KUKA KRL program: MyProgram_088().src

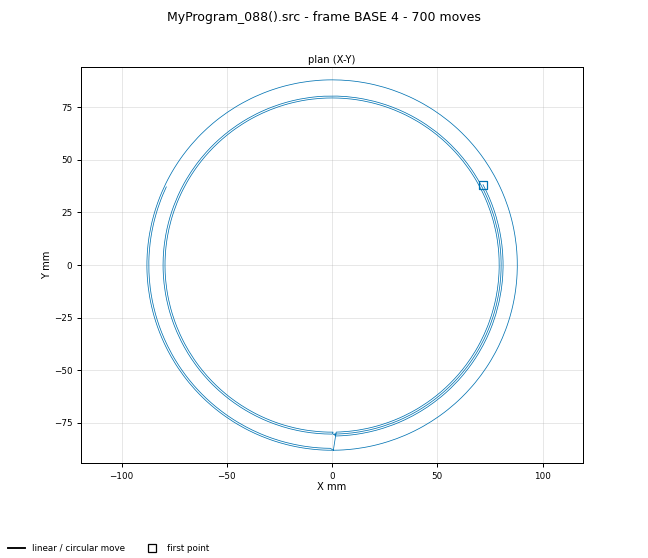
[picture p0: tool path of MyProgram_088().src in frame BASE 4, 700 of 700 moves have a stored position in this frame; points joined in program order, loops and branches not executed]
&ACCESS RVP
&REL 1
&PARAM TEMPLATE = C:\KRC\Roboter\Template\vorgabe
&PARAM EDITMASK = *
DEF MyProgram_088()
; ---- Setting reference (Base) ----
$BASE = BASE_DATA[4]

; --------------------------
; ---- Setting tool (TCP) ----
$TOOL = TOOL_DATA[3]
; --------------------------

$VEL.CP = VEL_APROX_PRINT
Startdeposition()
$VEL.CP = VEL_PRINT
LIN {X 71.7215,Y 38.1839,Z 85,A 22.0151,B 24.9008,C -2.2994,E1 25.1418,E2 422.6752} C_DIS
LIN {X 73.0397,Y 35.5985,Z 85,A 19.8506,B 24.9016,C -2.29,E1 25.1445,E2 424.8504} C_DIS
LIN {X 74.6096,Y 32.1771,Z 85,A 17.0372,B 24.9027,C -2.2774,E1 25.1477,E2 427.6781} C_DIS
LIN {X 75.8629,Y 29.0996,Z 85,A 14.4273,B 24.904,C -2.2622,E1 25.1504,E2 430.3095} C_DIS
LIN {X 77.0024,Y 25.9323,Z 85,A 12.4771,B 24.9034,C -2.2686,E1 25.1521,E2 432.2335} C_DIS
LIN {X 77.9339,Y 22.9819,Z 85,A 10.6782,B 24.903,C -2.2743,E1 25.1536,E2 434.0087} C_DIS
LIN {X 79.035,Y 18.8543,Z 85,A 7.5323,B 24.9041,C -2.2609,E1 25.1558,E2 437.1682} C_DIS
LIN {X 79.6807,Y 15.9069,Z 85,A 5.3667,B 24.9048,C -2.2531,E1 25.157,E2 439.3395} C_DIS
LIN {X 80.2365,Y 12.8106,Z 85,A 3.1294,B 24.9054,C -2.2456,E1 25.158,E2 441.5815} C_DIS
LIN {X 80.6846,Y 9.5848,Z 85,A 0.913,B 24.9058,C -2.241,E1 25.1588,E2 443.7957} C_DIS
LIN {X 81.034,Y 5.9647,Z 85,A -1.7315,B 24.9067,C -2.2303,E1 25.1595,E2 446.4497} C_DIS
LIN {X 81.2311,Y 1.8696,Z 85,A -4.5035,B 24.9071,C -2.2249,E1 25.1598,E2 449.2179} C_DIS
LIN {X 81.247,Y -1.0045,Z 85,A -6.6494,B 24.908,C -2.2146,E1 25.1598,E2 451.3753} C_DIS
LIN {X 81.1087,Y -4.833,Z 85,A -9.2665,B 24.9085,C -2.2087,E1 25.1594,E2 453.9908} C_DIS
LIN {X 80.8758,Y -7.8156,Z 85,A -11.3284,B 24.9089,C -2.2035,E1 25.1589,E2 456.0529} C_DIS
LIN {X 80.382,Y -11.8586,Z 85,A -14.402,B 24.9102,C -2.1879,E1 25.1577,E2 459.1452} C_DIS
LIN {X 79.3699,Y -17.3859,Z 85,A -18.0107,B 24.9103,C -2.1867,E1 25.1558,E2 462.7356} C_DIS
LIN {X 77.8059,Y -23.4136,Z 85,A -22.2752,B 24.9111,C -2.177,E1 25.1528,E2 466.9985} C_DIS
LIN {X 76.2109,Y -28.1759,Z 85,A -26.0321,B 24.9126,C -2.1591,E1 25.1493,E2 470.7765} C_DIS
LIN {X 74.9427,Y -31.3923,Z 85,A -28.361,B 24.9129,C -2.1552,E1 25.1469,E2 473.1018} C_DIS
LIN {X 73.4433,Y -34.7586,Z 85,A -31.6965,B 24.9154,C -2.1239,E1 25.1429,E2 476.4932} C_DIS
LIN {X 71.7565,Y -38.1174,Z 85,A -33.6164,B 24.9142,C -2.1394,E1 25.1405,E2 478.3663} C_DIS
LIN {X 69.6036,Y -41.9201,Z 85,A -36.6274,B 24.9147,C -2.1328,E1 25.1363,E2 481.3774} C_DIS
LIN {X 68.1735,Y -44.2082,Z 85,A -38.5092,B 24.9151,C -2.1281,E1 25.1334,E2 483.2608} C_DIS
LIN {X 66.6964,Y -46.4052,Z 85,A -40.2853,B 24.9152,C -2.1258,E1 25.1306,E2 485.0334} C_DIS
LIN {X 64.8908,Y -48.8983,Z 85,A -42.8716,B 24.9168,C -2.1068,E1 25.1263,E2 487.6524} C_DIS
LIN {X 62.174,Y -52.3114,Z 85,A -45.7058,B 24.9168,C -2.1064,E1 25.1213,E2 490.4744} C_DIS
LIN {X 59.9047,Y -54.8933,Z 85,A -48.3196,B 24.9177,C -2.0943,E1 25.1164,E2 493.1051} C_DIS
LIN {X 56.2805,Y -58.6036,Z 85,A -51.6653,B 24.9177,C -2.0953,E1 25.1098,E2 496.4343} C_DIS
LIN {X 53.8949,Y -60.8059,Z 85,A -54.008,B 24.9182,C -2.0883,E1 25.1049,E2 498.7841} C_DIS
LIN {X 51.8176,Y -62.5844,Z 85,A -56.0782,B 24.9189,C -2.0796,E1 25.1005,E2 500.867} C_DIS
LIN {X 48.3827,Y -65.2778,Z 85,A -59.0584,B 24.9192,C -2.0761,E1 25.0939,E2 503.8446} C_DIS
LIN {X 45.1916,Y -67.526,Z 85,A -61.807,B 24.9196,C -2.0707,E1 25.0875,E2 506.5965} C_DIS
LIN {X 41.9777,Y -69.5686,Z 85,A -64.4606,B 24.9199,C -2.0667,E1 25.0812,E2 509.2512} C_DIS
LIN {X 38.2675,Y -71.6774,Z 85,A -67.1339,B 24.9195,C -2.0718,E1 25.0748,E2 511.9045} C_DIS
LIN {X 34.642,Y -73.4979,Z 85,A -69.9393,B 24.9197,C -2.0688,E1 25.0678,E2 514.7094} C_DIS
LIN {X 32.2174,Y -74.592,Z 85,A -72.1455,B 24.9207,C -2.0559,E1 25.062,E2 516.9409} C_DIS
LIN {X 29.1592,Y -75.8403,Z 85,A -75.5951,B 24.9236,C -2.0189,E1 25.0529,E2 520.4705} C_DIS
LIN {X 24.2438,Y -77.5508,Z 85,A -77.6595,B 24.9202,C -2.0628,E1 25.0477,E2 522.427} C_DIS
LIN {X 21.102,Y -78.4638,Z 85,A -80.9066,B 24.9226,C -2.032,E1 25.0387,E2 525.7419} C_DIS
LIN {X 17.9007,Y -79.2564,Z 85,A -82.7247,B 24.9216,C -2.0449,E1 25.0339,E2 527.5267} C_DIS
LIN {X 14.15,Y -80.0105,Z 85,A -85.3692,B 24.9216,C -2.0443,E1 25.0266,E2 530.1696} C_DIS
LIN {X 11.1964,Y -80.477,Z 85,A -87.4429,B 24.9216,C -2.0439,E1 25.0209,E2 532.2425} C_DIS
LIN {X 8.4006,Y -80.8164,Z 85,A -89.3615,B 24.9216,C -2.0447,E1 25.0156,E2 534.1577} C_DIS
LIN {X 4.7091,Y -81.1155,Z 85,A -92.0431,B 24.9219,C -2.0414,E1 25.0081,E2 536.8458} C_DIS
LIN {X 1.9082,Y -81.2304,Z 85,A -94.1506,B 24.9222,C -2.0369,E1 25.0022,E2 538.9635} C_DIS
LIN {X 1.9082,Y -81.2304,Z 85,A -94.1506,B 24.9222,C -2.0369,E1 25.0022,E2 538.9635} C_DIS
Enddeposition()
LIN {X 0.4892,Y -80.3266,Z 85,A -94.3055,B 24.919,C -2.0777,E1 25.002,E2 539.0217} C_DIS
Startdeposition()
$VEL.CP = VEL_PRINT
LIN {X 3.1515,Y -80.2693,Z 85,A -92.135,B 24.9184,C -2.0862,E1 25.0081,E2 536.8314} C_DIS
LIN {X 6.3093,Y -80.0825,Z 85,A -89.8012,B 24.9181,C -2.0896,E1 25.0147,E2 534.4908} C_DIS
LIN {X 9.7464,Y -79.7382,Z 85,A -87.3488,B 24.9181,C -2.0906,E1 25.0215,E2 532.0375} C_DIS
LIN {X 13.0866,Y -79.2576,Z 85,A -85.1111,B 24.9183,C -2.0873,E1 25.0276,E2 529.8099} C_DIS
LIN {X 17.5265,Y -78.3964,Z 85,A -81.2162,B 24.9165,C -2.1104,E1 25.0384,E2 525.8651} C_DIS
LIN {X 20.7087,Y -77.6158,Z 85,A -78.875,B 24.9163,C -2.113,E1 25.0447,E2 523.5215} C_DIS
LIN {X 23.9024,Y -76.6922,Z 85,A -77.0409,B 24.9174,C -2.0993,E1 25.0495,E2 521.7232} C_DIS
LIN {X 28.6458,Y -75.0497,Z 85,A -73.465,B 24.917,C -2.1037,E1 25.0589,E2 518.144} C_DIS
LIN {X 31.5046,Y -73.8957,Z 85,A -71.3926,B 24.917,C -2.103,E1 25.0643,E2 516.0783} C_DIS
LIN {X 33.8559,Y -72.8477,Z 85,A -69.6419,B 24.917,C -2.1032,E1 25.0687,E2 514.3314} C_DIS
LIN {X 37.6269,Y -70.9737,Z 85,A -66.9168,B 24.9173,C -2.0995,E1 25.0755,E2 511.6225} C_DIS
LIN {X 40.5219,Y -69.3625,Z 85,A -64.1229,B 24.9159,C -2.117,E1 25.0823,E2 508.7954} C_DIS
LIN {X 43.3163,Y -67.6514,Z 85,A -61.8824,B 24.9159,C -2.1184,E1 25.0876,E2 506.5587} C_DIS
LIN {X 46.0185,Y -65.8433,Z 85,A -59.5276,B 24.9154,C -2.1242,E1 25.0931,E2 504.1983} C_DIS
LIN {X 48.3059,Y -64.1837,Z 85,A -57.4844,B 24.915,C -2.1292,E1 25.0977,E2 502.1505} C_DIS
LIN {X 50.7678,Y -62.2551,Z 85,A -55.2771,B 24.9146,C -2.1333,E1 25.1025,E2 499.9417} C_DIS
LIN {X 53.1527,Y -60.2326,Z 85,A -53.0638,B 24.9143,C -2.1378,E1 25.1071,E2 497.7265} C_DIS
LIN {X 55.3912,Y -58.1813,Z 85,A -50.8101,B 24.9136,C -2.1457,E1 25.1118,E2 495.4634} C_DIS
LIN {X 57.8412,Y -55.7441,Z 85,A -48.6116,B 24.9138,C -2.1433,E1 25.116,E2 493.2801} C_DIS
LIN {X 59.663,Y -53.7904,Z 85,A -46.5788,B 24.9131,C -2.1521,E1 25.1199,E2 491.2354} C_DIS
LIN {X 61.6699,Y -51.4768,Z 85,A -44.4422,B 24.9128,C -2.1562,E1 25.1238,E2 489.0988} C_DIS
LIN {X 63.5272,Y -49.1663,Z 85,A -42.3702,B 24.9125,C -2.1604,E1 25.1273,E2 487.0266} C_DIS
LIN {X 64.9007,Y -47.3384,Z 85,A -40.6906,B 24.912,C -2.1664,E1 25.1301,E2 485.341} C_DIS
LIN {X 66.6996,Y -44.7691,Z 85,A -38.3931,B 24.9113,C -2.1745,E1 25.1338,E2 483.0356} C_DIS
LIN {X 68.4937,Y -41.9727,Z 85,A -36.1059,B 24.911,C -2.1785,E1 25.1372,E2 480.7504} C_DIS
LIN {X 70.1605,Y -39.1217,Z 85,A -33.8246,B 24.9106,C -2.183,E1 25.1403,E2 478.4705} C_DIS
LIN {X 72.1071,Y -35.4071,Z 85,A -30.886,B 24.91,C -2.19,E1 25.1441,E2 475.5308} C_DIS
LIN {X 73.2284,Y -33.0244,Z 85,A -29.0291,B 24.9096,C -2.195,E1 25.1462,E2 473.6722} C_DIS
LIN {X 74.3269,Y -30.4722,Z 85,A -27.0214,B 24.9091,C -2.2018,E1 25.1484,E2 471.6595} C_DIS
LIN {X 75.3494,Y -27.8495,Z 85,A -25.0113,B 24.9085,C -2.208,E1 25.1504,E2 469.6459} C_DIS
LIN {X 76.4207,Y -24.7565,Z 85,A -22.8102,B 24.9083,C -2.2109,E1 25.1524,E2 467.4503} C_DIS
LIN {X 77.1844,Y -22.2647,Z 85,A -20.0818,B 24.9054,C -2.2451,E1 25.1546,E2 464.657} C_DIS
LIN {X 78.1334,Y -18.6635,Z 85,A -18.1352,B 24.9067,C -2.2302,E1 25.1558,E2 462.7566} C_DIS
LIN {X 79.0955,Y -14.0334,Z 85,A -14.2314,B 24.9043,C -2.2583,E1 25.1579,E2 458.8094} C_DIS
LIN {X 79.6066,Y -10.7628,Z 85,A -12.706,B 24.906,C -2.2386,E1 25.1585,E2 457.3395} C_DIS
LIN {X 79.8247,Y -9.0073,Z 85,A -11.1445,B 24.9048,C -2.2523,E1 25.159,E2 455.7547} C_DIS
LIN {X 80.1211,Y -5.8107,Z 85,A -8.9024,B 24.9043,C -2.2581,E1 25.1595,E2 453.5123} C_DIS
LIN {X 80.2889,Y -2.5914,Z 85,A -6.6753,B 24.9039,C -2.2631,E1 25.1597,E2 451.2866} C_DIS
LIN {X 80.328,Y 0.73,Z 85,A -4.1962,B 24.903,C -2.2742,E1 25.1597,E2 448.7961} C_DIS
LIN {X 80.228,Y 4.074,Z 85,A -1.9038,B 24.9026,C -2.2788,E1 25.1595,E2 446.5066} C_DIS
LIN {X 79.9921,Y 7.3672,Z 85,A 0.4357,B 24.902,C -2.2857,E1 25.1589,E2 444.1645} C_DIS
LIN {X 79.6182,Y 10.6808,Z 85,A 2.8385,B 24.9013,C -2.294,E1 25.1581,E2 441.7564} C_DIS
LIN {X 79.1715,Y 13.6013,Z 85,A 4.9208,B 24.9008,C -2.2997,E1 25.1572,E2 439.6727} C_DIS
LIN {X 78.5178,Y 16.97,Z 85,A 7.2722,B 24.9004,C -2.3042,E1 25.1559,E2 437.3245} C_DIS
LIN {X 76.8809,Y 23.2925,Z 85,A 11.7016,B 24.8998,C -2.3108,E1 25.1527,E2 432.9049} C_DIS
LIN {X 74.9629,Y 28.8753,Z 85,A 16.0802,B 24.8983,C -2.3285,E1 25.1486,E2 428.5091} C_DIS
LIN {X 73.7475,Y 31.8495,Z 85,A 18.4097,B 24.8976,C -2.3363,E1 25.1461,E2 426.174} C_DIS
LIN {X 72.3676,Y 34.8703,Z 85,A 20.7576,B 24.8971,C -2.3423,E1 25.1433,E2 423.8246} C_DIS
LIN {X 71.0185,Y 37.5418,Z 85,A 22.8625,B 24.8966,C -2.3472,E1 25.1406,E2 421.7193} C_DIS
LIN {X 69.3238,Y 40.5873,Z 85,A 25.4545,B 24.8957,C -2.3572,E1 25.137,E2 419.1172} C_DIS
LIN {X 67.5519,Y 43.4713,Z 85,A 27.7924,B 24.8954,C -2.361,E1 25.1335,E2 416.782} C_DIS
LIN {X 66.1104,Y 45.6344,Z 85,A 29.5804,B 24.8952,C -2.3636,E1 25.1307,E2 414.9967} C_DIS
LIN {X 64.1702,Y 48.3239,Z 85,A 31.7935,B 24.8951,C -2.3646,E1 25.127,E2 412.792} C_DIS
LIN {X 62.1138,Y 50.9421,Z 85,A 34.0874,B 24.8948,C -2.3676,E1 25.1231,E2 410.5015} C_DIS
LIN {X 59.6325,Y 53.8245,Z 85,A 38.0034,B 24.8909,C -2.4116,E1 25.1156,E2 406.4989} C_DIS
LIN {X 56.4551,Y 57.1474,Z 85,A 40.0383,B 24.8937,C -2.3796,E1 25.1118,E2 404.5486} C_DIS
LIN {X 54.5173,Y 58.9995,Z 85,A 42.1754,B 24.8928,C -2.3904,E1 25.1074,E2 402.3946} C_DIS
LIN {X 51.3663,Y 61.7617,Z 85,A 44.9754,B 24.8928,C -2.3904,E1 25.1015,E2 399.6057} C_DIS
LIN {X 49.3377,Y 63.3951,Z 85,A 46.9941,B 24.892,C -2.3987,E1 25.097,E2 397.5748} C_DIS
LIN {X 44.6406,Y 66.7866,Z 85,A 50.9065,B 24.892,C -2.3988,E1 25.0882,E2 393.6756} C_DIS
LIN {X 42.4805,Y 68.1793,Z 85,A 52.8244,B 24.8915,C -2.4043,E1 25.0836,E2 391.7511} C_DIS
LIN {X 40.1164,Y 69.5966,Z 85,A 54.8115,B 24.8912,C -2.4077,E1 25.0788,E2 389.7618} C_DIS
LIN {X 37.418,Y 71.0837,Z 85,A 57.0852,B 24.8907,C -2.413,E1 25.0732,E2 387.4821} C_DIS
LIN {X 34.7082,Y 72.4455,Z 85,A 59.2334,B 24.8905,C -2.4152,E1 25.0679,E2 385.3344} C_DIS
LIN {X 31.6701,Y 73.8257,Z 85,A 61.6846,B 24.8901,C -2.4199,E1 25.0616,E2 382.878} C_DIS
LIN {X 28.64,Y 75.052,Z 85,A 63.8969,B 24.8902,C -2.4187,E1 25.0558,E2 380.6736} C_DIS
LIN {X 25.7053,Y 76.1068,Z 85,A 66.0778,B 24.8902,C -2.4193,E1 25.0501,E2 378.4955} C_DIS
LIN {X 22.0903,Y 77.2338,Z 85,A 68.4644,B 24.8908,C -2.412,E1 25.0438,E2 376.1304} C_DIS
LIN {X 19.8866,Y 77.8302,Z 85,A 70.9808,B 24.8883,C -2.4392,E1 25.0368,E2 373.5534} C_DIS
LIN {X 14.8968,Y 78.9378,Z 85,A 74.3625,B 24.8889,C -2.433,E1 25.0276,E2 370.1906} C_DIS
LIN {X 11.5765,Y 79.4926,Z 85,A 77.5311,B 24.8868,C -2.4563,E1 25.0187,E2 366.9697} C_DIS
LIN {X 7.0031,Y 80.0257,Z 85,A 79.5681,B 24.8901,C -2.4203,E1 25.0133,E2 365.0194} C_DIS
LIN {X 2.4401,Y 80.2935,Z 85,A 82.9335,B 24.8898,C -2.4232,E1 25.0039,E2 361.6484} C_DIS
LIN {X -3.8247,Y 80.2404,Z 85,A 87.5593,B 24.8895,C -2.4264,E1 24.991,E2 357.0144} C_DIS
LIN {X -7.0125,Y 80.0248,Z 85,A 89.8582,B 24.8895,C -2.426,E1 24.9846,E2 354.7156} C_DIS
LIN {X -10.2057,Y 79.6797,Z 85,A 92.0577,B 24.8899,C -2.4221,E1 24.9785,E2 352.5238} C_DIS
LIN {X -15.2017,Y 78.8791,Z 85,A 95.701,B 24.8901,C -2.4205,E1 24.9685,E2 348.8809} C_DIS
LIN {X -18.5339,Y 78.1647,Z 85,A 98.1174,B 24.8903,C -2.4179,E1 24.9619,E2 346.4676} C_DIS
LIN {X -21.4983,Y 77.4016,Z 85,A 100.3804,B 24.8903,C -2.4179,E1 24.9558,E2 344.2012} C_DIS
LIN {X -24.6371,Y 76.4593,Z 85,A 103.1487,B 24.8894,C -2.4272,E1 24.9483,E2 341.4059} C_DIS
LIN {X -28.7937,Y 74.9937,Z 85,A 105.8355,B 24.891,C -2.4105,E1 24.9414,E2 338.7532} C_DIS
LIN {X -30.8196,Y 74.1844,Z 85,A 107.448,B 24.891,C -2.4099,E1 24.9372,E2 337.1386} C_DIS
LIN {X -33.7994,Y 72.874,Z 85,A 109.6874,B 24.8915,C -2.4042,E1 24.9315,E2 334.9073} C_DIS
LIN {X -36.0699,Y 71.7785,Z 85,A 111.9608,B 24.8906,C -2.4143,E1 24.9258,E2 332.6039} C_DIS
LIN {X -40.0277,Y 69.6476,Z 85,A 114.6461,B 24.8924,C -2.3947,E1 24.9193,E2 329.9576} C_DIS
LIN {X -42.3641,Y 68.252,Z 85,A 116.6645,B 24.8925,C -2.3932,E1 24.9145,E2 327.9364} C_DIS
LIN {X -44.9874,Y 66.5518,Z 85,A 119.9044,B 24.8904,C -2.4162,E1 24.9069,E2 324.6309} C_DIS
LIN {X -48.6045,Y 63.9594,Z 85,A 122.2733,B 24.893,C -2.3879,E1 24.9017,E2 322.321} C_DIS
LIN {X -51.0902,Y 61.9911,Z 85,A 124.4404,B 24.8937,C -2.3805,E1 24.897,E2 320.1635} C_DIS
LIN {X -53.6223,Y 59.8135,Z 85,A 126.6786,B 24.8945,C -2.3713,E1 24.8923,E2 317.9383} C_DIS
LIN {X -55.7888,Y 57.7981,Z 85,A 128.8046,B 24.8949,C -2.3668,E1 24.888,E2 315.8142} C_DIS
LIN {X -57.81,Y 55.7765,Z 85,A 130.909,B 24.8952,C -2.3636,E1 24.8839,E2 313.7085} C_DIS
LIN {X -59.9727,Y 53.4445,Z 85,A 133.3311,B 24.8953,C -2.362,E1 24.8793,E2 311.2795} C_DIS
LIN {X -62.2163,Y 50.8156,Z 85,A 135.7691,B 24.8959,C -2.355,E1 24.875,E2 308.8471} C_DIS
LIN {X -64.4386,Y 47.9666,Z 85,A 138.113,B 24.8971,C -2.3421,E1 24.871,E2 306.5229} C_DIS
LIN {X -66.8386,Y 44.5599,Z 85,A 141.51,B 24.8968,C -2.345,E1 24.8656,E2 303.1021} C_DIS
LIN {X -69.1601,Y 40.8643,Z 85,A 144.0739,B 24.8988,C -2.322,E1 24.8619,E2 300.58} C_DIS
LIN {X -70.4174,Y 38.6595,Z 85,A 146.39,B 24.8982,C -2.3298,E1 24.8587,E2 298.233} C_DIS
LIN {X -71.8855,Y 35.8542,Z 85,A 148.7868,B 24.8984,C -2.3268,E1 24.8557,E2 295.8306} C_DIS
LIN {X -73.222,Y 33.0385,Z 85,A 152.0244,B 24.8967,C -2.3467,E1 24.8519,E2 292.5277} C_DIS
LIN {X -75.2268,Y 28.1783,Z 85,A 154.3321,B 24.9009,C -2.2977,E1 24.8497,E2 290.324} C_DIS
LIN {X -76.065,Y 25.8294,Z 85,A 156.3338,B 24.9009,C -2.298,E1 24.8478,E2 288.3103} C_DIS
LIN {X -76.9901,Y 22.9246,Z 85,A 158.4714,B 24.9016,C -2.2903,E1 24.8461,E2 286.1787} C_DIS
LIN {X -77.7783,Y 20.0887,Z 85,A 160.6209,B 24.902,C -2.285,E1 24.8445,E2 284.0293} C_DIS
LIN {X -78.4855,Y 17.1181,Z 85,A 162.824,B 24.9026,C -2.2788,E1 24.8432,E2 281.8282} C_DIS
LIN {X -79.0714,Y 14.1674,Z 85,A 165.0081,B 24.9031,C -2.273,E1 24.842,E2 279.645} C_DIS
LIN {X -79.6634,Y 10.3317,Z 85,A 167.6424,B 24.9041,C -2.2608,E1 24.841,E2 277.0243} C_DIS
LIN {X -79.9716,Y 7.5891,Z 85,A 170.6028,B 24.9025,C -2.2801,E1 24.8402,E2 274} C_DIS
LIN {X -80.2497,Y 3.6068,Z 85,A 172.3641,B 24.9056,C -2.243,E1 24.8399,E2 272.3166} C_DIS
LIN {X -80.3321,Y 0.0663,Z 85,A 174.9252,B 24.9062,C -2.2358,E1 24.8398,E2 269.7573} C_DIS
LIN {X -80.2998,Y -2.2362,Z 85,A 176.7532,B 24.9062,C -2.2353,E1 24.8398,E2 267.9194} C_DIS
LIN {X -80.1663,Y -5.1424,Z 85,A 178.9332,B 24.9066,C -2.2314,E1 24.8402,E2 265.7356} C_DIS
LIN {X -79.8482,Y -8.8017,Z 85,A -178.2385,B 24.9068,C -2.2285,E1 24.841,E2 262.8972} C_DIS
LIN {X -79.2484,Y -13.1416,Z 85,A -175.2705,B 24.908,C -2.2148,E1 24.8422,E2 259.9445} C_DIS
LIN {X -78.6741,Y -16.2293,Z 85,A -172.7035,B 24.9079,C -2.2163,E1 24.8436,E2 257.3585} C_DIS
LIN {X -77.7492,Y -20.2018,Z 85,A -170.3797,B 24.9098,C -2.1923,E1 24.8451,E2 255.0784} C_DIS
LIN {X -77.1874,Y -22.2543,Z 85,A -168.4168,B 24.9093,C -2.1992,E1 24.8467,E2 253.0877} C_DIS
LIN {X -76.1655,Y -25.5312,Z 85,A -166.1295,B 24.9102,C -2.1878,E1 24.8486,E2 250.8145} C_DIS
LIN {X -75.154,Y -28.3707,Z 85,A -163.8802,B 24.9105,C -2.1841,E1 24.8508,E2 248.5613} C_DIS
LIN {X -73.8881,Y -31.5228,Z 85,A -161.0025,B 24.9101,C -2.1891,E1 24.8539,E2 245.6557} C_DIS
LIN {X -71.7089,Y -36.2077,Z 85,A -157.7774,B 24.9119,C -2.1668,E1 24.8578,E2 242.4664} C_DIS
LIN {X -70.252,Y -38.9578,Z 85,A -154.9226,B 24.9111,C -2.1776,E1 24.8617,E2 239.5707} C_DIS
LIN {X -68.5214,Y -41.9271,Z 85,A -153.135,B 24.913,C -2.1536,E1 24.8642,E2 237.8313} C_DIS
LIN {X -66.831,Y -44.5736,Z 85,A -150.6758,B 24.913,C -2.1537,E1 24.868,E2 235.3595} C_DIS
LIN {X -64.5591,Y -47.805,Z 85,A -147.9959,B 24.9139,C -2.1431,E1 24.8723,E2 232.6917} C_DIS
LIN {X -62.834,Y -50.0498,Z 85,A -146.0042,B 24.9143,C -2.1376,E1 24.8758,E2 230.7038} C_DIS
LIN {X -61.0021,Y -52.2666,Z 85,A -144.0636,B 24.9149,C -2.13,E1 24.8792,E2 228.7725} C_DIS
LIN {X -58.6328,Y -54.9111,Z 85,A -141.4752,B 24.9152,C -2.1259,E1 24.8841,E2 226.1825} C_DIS
LIN {X -56.6063,Y -56.9981,Z 85,A -139.0227,B 24.9148,C -2.1317,E1 24.889,E2 223.7056} C_DIS
LIN {X -54.019,Y -59.4568,Z 85,A -136.6705,B 24.9156,C -2.1213,E1 24.8938,E2 221.3686} C_DIS
LIN {X -51.559,Y -61.6016,Z 85,A -134.3702,B 24.916,C -2.1162,E1 24.8986,E2 219.0716} C_DIS
LIN {X -49.1018,Y -63.577,Z 85,A -131.8396,B 24.9157,C -2.1199,E1 24.9043,E2 216.5229} C_DIS
LIN {X -46.4747,Y -65.5222,Z 85,A -129.7172,B 24.9165,C -2.1102,E1 24.909,E2 214.4162} C_DIS
LIN {X -43.7958,Y -67.3436,Z 85,A -127.452,B 24.9169,C -2.1053,E1 24.9143,E2 212.1552} C_DIS
LIN {X -41.2543,Y -68.9293,Z 85,A -125.4521,B 24.9174,C -2.0984,E1 24.919,E2 210.1655} C_DIS
LIN {X -39.1467,Y -70.1466,Z 85,A -122.9713,B 24.916,C -2.1168,E1 24.9252,E2 207.6336} C_DIS
LIN {X -36.1217,Y -71.7521,Z 85,A -120.4266,B 24.916,C -2.1167,E1 24.9316,E2 205.0825} C_DIS
LIN {X -32.8319,Y -73.3151,Z 85,A -118.7548,B 24.9183,C -2.0877,E1 24.9357,E2 203.4756} C_DIS
LIN {X -30.4489,Y -74.3364,Z 85,A -116.7428,B 24.9181,C -2.0904,E1 24.9409,E2 201.4526} C_DIS
LIN {X -27.7567,Y -75.3832,Z 85,A -114.2267,B 24.9172,C -2.1014,E1 24.9475,E2 198.9049} C_DIS
LIN {X -23.5857,Y -76.7904,Z 85,A -111.2646,B 24.9178,C -2.094,E1 24.9554,E2 195.9553} C_DIS
LIN {X -19.9178,Y -77.8222,Z 85,A -108.0406,B 24.9167,C -2.107,E1 24.9642,E2 192.6955} C_DIS
LIN {X -16.3419,Y -78.651,Z 85,A -106.184,B 24.9186,C -2.0838,E1 24.9691,E2 190.8919} C_DIS
LIN {X -13.2932,Y -79.2231,Z 85,A -103.8794,B 24.9184,C -2.0857,E1 24.9754,E2 188.5803} C_DIS
LIN {X -10.0367,Y -79.7016,Z 85,A -101.5179,B 24.9184,C -2.0857,E1 24.982,E2 186.2172} C_DIS
LIN {X -6.7325,Y -80.0487,Z 85,A -99.1532,B 24.9184,C -2.0853,E1 24.9886,E2 183.8521} C_DIS
LIN {X -3.5295,Y -80.2531,Z 85,A -96.8148,B 24.9184,C -2.0869,E1 24.9951,E2 181.5092} C_DIS
LIN {X -0.0125,Y -80.332,Z 85,A -94.327,B 24.9184,C -2.0867,E1 25.002,E2 179.0217} C_DIS
LIN {X -0.0125,Y -80.332,Z 85,A -94.327,B 24.9184,C -2.0867,E1 25.002,E2 179.0217} C_DIS
Enddeposition()
LIN {X 0.4836,Y -79.4079,Z 85,A -94.5866,B 24.9184,C -2.0848,E1 25.0013,E2 179.2858} C_DIS
Startdeposition()
$VEL.CP = VEL_PRINT
LIN {X -2.023,Y -79.3847,Z 85,A -96.676,B 24.9191,C -2.0764,E1 24.9954,E2 181.3953} C_DIS
LIN {X -4.2492,Y -79.2958,Z 85,A -98.501,B 24.9196,C -2.0701,E1 24.9903,E2 183.2357} C_DIS
LIN {X -6.819,Y -79.1176,Z 85,A -100.2396,B 24.9194,C -2.0735,E1 24.9855,E2 184.967} C_DIS
LIN {X -8.756,Y -78.9267,Z 85,A -101.5959,B 24.9193,C -2.075,E1 24.9817,E2 186.3204} C_DIS
LIN {X -10.7645,Y -78.6775,Z 85,A -103.0049,B 24.9191,C -2.0767,E1 24.9778,E2 187.7264} C_DIS
LIN {X -12.6896,Y -78.39,Z 85,A -104.413,B 24.9191,C -2.077,E1 24.9739,E2 189.1351} C_DIS
LIN {X -15.1166,Y -77.9574,Z 85,A -106.4091,B 24.9195,C -2.0715,E1 24.9684,E2 191.1463} C_DIS
LIN {X -18.1449,Y -77.3091,Z 85,A -108.5779,B 24.9193,C -2.0744,E1 24.9625,E2 193.3109} C_DIS
LIN {X -20.3474,Y -76.7592,Z 85,A -110.0636,B 24.9189,C -2.0796,E1 24.9585,E2 194.7866} C_DIS
LIN {X -22.2087,Y -76.2416,Z 85,A -111.5113,B 24.9189,C -2.079,E1 24.9546,E2 196.238} C_DIS
LIN {X -24.4792,Y -75.5422,Z 85,A -113.3856,B 24.9192,C -2.0758,E1 24.9496,E2 198.123} C_DIS
LIN {X -26.7593,Y -74.7665,Z 85,A -115.0209,B 24.9189,C -2.0801,E1 24.9453,E2 199.7514} C_DIS
LIN {X -28.6537,Y -74.0607,Z 85,A -116.6432,B 24.9191,C -2.077,E1 24.941,E2 201.3846} C_DIS
LIN {X -31.2912,Y -72.986,Z 85,A -118.4944,B 24.9185,C -2.0846,E1 24.9363,E2 203.2218} C_DIS
LIN {X -33.5785,Y -71.9607,Z 85,A -120.4844,B 24.9187,C -2.0817,E1 24.9312,E2 205.2237} C_DIS
LIN {X -35.8052,Y -70.8801,Z 85,A -122.0759,B 24.9182,C -2.0891,E1 24.9273,E2 206.8017} C_DIS
LIN {X -37.5425,Y -69.9753,Z 85,A -123.5424,B 24.9182,C -2.0895,E1 24.9236,E2 208.2714} C_DIS
LIN {X -39.994,Y -68.6044,Z 85,A -125.5478,B 24.9179,C -2.0928,E1 24.9188,E2 210.2747} C_DIS
LIN {X -41.7274,Y -67.5637,Z 85,A -126.9591,B 24.9176,C -2.0963,E1 24.9154,E2 211.6822} C_DIS
LIN {X -43.3047,Y -66.5643,Z 85,A -128.5942,B 24.918,C -2.0906,E1 24.9115,E2 213.336} C_DIS
LIN {X -45.9316,Y -64.7781,Z 85,A -130.8638,B 24.9177,C -2.095,E1 24.9063,E2 215.603} C_DIS
LIN {X -48.4803,Y -62.8929,Z 85,A -133.0733,B 24.9172,C -2.101,E1 24.9014,E2 217.8059} C_DIS
LIN {X -50.7858,Y -61.0464,Z 85,A -135.2329,B 24.917,C -2.1042,E1 24.8967,E2 219.9662} C_DIS
LIN {X -52.9638,Y -59.1667,Z 85,A -137.2967,B 24.9166,C -2.1085,E1 24.8924,E2 222.0278} C_DIS
LIN {X -55.0999,Y -57.1827,Z 85,A -139.4379,B 24.9164,C -2.1118,E1 24.888,E2 224.17} C_DIS
LIN {X -57.1753,Y -55.1076,Z 85,A -141.5707,B 24.916,C -2.1159,E1 24.8839,E2 226.3022} C_DIS
LIN {X -59.4381,Y -52.6606,Z 85,A -144.0868,B 24.9158,C -2.1183,E1 24.8791,E2 228.8238} C_DIS
LIN {X -61.4124,Y -50.3445,Z 85,A -146.2496,B 24.9154,C -2.1242,E1 24.8753,E2 230.9824} C_DIS
LIN {X -63.1958,Y -48.0872,Z 85,A -148.1826,B 24.9147,C -2.1328,E1 24.872,E2 232.904} C_DIS
LIN {X -64.3986,Y -46.4634,Z 85,A -149.5579,B 24.9142,C -2.1385,E1 24.8697,E2 234.2724} C_DIS
LIN {X -65.6387,Y -44.6929,Z 85,A -151.3685,B 24.9144,C -2.136,E1 24.8668,E2 236.0979} C_DIS
LIN {X -67.2326,Y -42.2573,Z 85,A -153.1943,B 24.9134,C -2.1483,E1 24.8641,E2 237.9034} C_DIS
LIN {X -68.1675,Y -40.7332,Z 85,A -154.5271,B 24.9133,C -2.1506,E1 24.8622,E2 239.2376} C_DIS
LIN {X -69.1409,Y -39.0583,Z 85,A -155.9331,B 24.913,C -2.1541,E1 24.8602,E2 240.6427} C_DIS
LIN {X -70.0738,Y -37.3588,Z 85,A -157.4274,B 24.9129,C -2.1554,E1 24.8582,E2 242.1417} C_DIS
LIN {X -71.0193,Y -35.5275,Z 85,A -158.8128,B 24.9123,C -2.1621,E1 24.8565,E2 243.5186} C_DIS
LIN {X -72.1907,Y -33.0844,Z 85,A -160.8938,B 24.9121,C -2.1643,E1 24.854,E2 245.6055} C_DIS
LIN {X -73.018,Y -31.2153,Z 85,A -162.3424,B 24.9117,C -2.1692,E1 24.8524,E2 247.0506} C_DIS
LIN {X -73.7328,Y -29.4884,Z 85,A -163.9737,B 24.912,C -2.1659,E1 24.8507,E2 248.6987} C_DIS
LIN {X -74.774,Y -26.7382,Z 85,A -165.9217,B 24.9111,C -2.1765,E1 24.8488,E2 250.6326} C_DIS
LIN {X -75.4297,Y -24.827,Z 85,A -167.2494,B 24.9105,C -2.184,E1 24.8476,E2 251.9498} C_DIS
LIN {X -75.9927,Y -23.0476,Z 85,A -168.8674,B 24.9108,C -2.1812,E1 24.8463,E2 253.5838} C_DIS
LIN {X -76.7876,Y -20.2425,Z 85,A -170.8446,B 24.91,C -2.1907,E1 24.8448,E2 255.5498} C_DIS
LIN {X -77.2856,Y -18.2464,Z 85,A -172.2171,B 24.9094,C -2.1981,E1 24.8439,E2 256.9128} C_DIS
LIN {X -77.6927,Y -16.4293,Z 85,A -173.6697,B 24.9093,C -2.1995,E1 24.843,E2 258.3707} C_DIS
LIN {X -78.0847,Y -14.4499,Z 85,A -175.2582,B 24.9092,C -2.2006,E1 24.8422,E2 259.9657} C_DIS
LIN {X -78.5511,Y -11.6541,Z 85,A -177.2298,B 24.9085,C -2.2088,E1 24.8414,E2 261.9295} C_DIS
LIN {X -78.8263,Y -9.6134,Z 85,A -178.5915,B 24.9078,C -2.2166,E1 24.8409,E2 263.2809} C_DIS
LIN {X -79.0376,Y -7.6858,Z 85,A 179.9996,B 24.9075,C -2.2207,E1 24.8405,E2 264.6882} C_DIS
LIN {X -79.2018,Y -5.7522,Z 85,A 178.5898,B 24.9071,C -2.2249,E1 24.8402,E2 266.0966} C_DIS
LIN {X -79.3412,Y -3.294,Z 85,A 176.6763,B 24.907,C -2.2271,E1 24.8399,E2 268.0163} C_DIS
LIN {X -79.4093,Y -0.3971,Z 85,A 174.4927,B 24.9066,C -2.2315,E1 24.8398,E2 270.2027} C_DIS
LIN {X -79.3844,Y 2.0334,Z 85,A 172.9295,B 24.9057,C -2.2418,E1 24.8398,E2 271.7507} C_DIS
LIN {X -79.309,Y 4.0099,Z 85,A 171.4924,B 24.9054,C -2.2461,E1 24.84,E2 273.1862} C_DIS
LIN {X -79.1879,Y 5.9405,Z 85,A 170.0866,B 24.905,C -2.2503,E1 24.8403,E2 274.5903} C_DIS
LIN {X -78.9547,Y 8.4885,Z 85,A 168.0489,B 24.905,C -2.2514,E1 24.8408,E2 276.6376} C_DIS
LIN {X -78.6094,Y 11.2439,Z 85,A 166.0171,B 24.9044,C -2.2571,E1 24.8416,E2 278.668} C_DIS
LIN {X -78.2399,Y 13.5867,Z 85,A 164.4314,B 24.9037,C -2.2656,E1 24.8423,E2 280.2427} C_DIS
LIN {X -77.8683,Y 15.5741,Z 85,A 162.9618,B 24.9033,C -2.27,E1 24.8431,E2 281.7106} C_DIS
LIN {X -77.481,Y 17.4009,Z 85,A 161.605,B 24.903,C -2.274,E1 24.8439,E2 283.0658} C_DIS
LIN {X -77.0124,Y 19.3681,Z 85,A 160.1357,B 24.9026,C -2.2783,E1 24.8449,E2 284.5334} C_DIS
LIN {X -76.536,Y 21.1737,Z 85,A 158.7336,B 24.9024,C -2.2812,E1 24.8459,E2 285.9368} C_DIS
LIN {X -75.9719,Y 23.1151,Z 85,A 157.3538,B 24.9018,C -2.2877,E1 24.847,E2 287.309} C_DIS
LIN {X -75.2264,Y 25.4332,Z 85,A 155.45,B 24.9017,C -2.2895,E1 24.8486,E2 289.2194} C_DIS
LIN {X -74.3766,Y 27.8222,Z 85,A 153.71,B 24.901,C -2.2973,E1 24.8503,E2 290.9507} C_DIS
LIN {X -73.7152,Y 29.5315,Z 85,A 152.3404,B 24.9007,C -2.3001,E1 24.8517,E2 292.3212} C_DIS
LIN {X -72.9794,Y 31.3061,Z 85,A 150.93,B 24.9004,C -2.3037,E1 24.8532,E2 293.7308} C_DIS
LIN {X -71.7797,Y 33.9669,Z 85,A 148.8525,B 24.8998,C -2.3107,E1 24.8556,E2 295.8031} C_DIS
LIN {X -70.9277,Y 35.712,Z 85,A 147.442,B 24.8995,C -2.3145,E1 24.8574,E2 297.2119} C_DIS
LIN {X -69.9701,Y 37.5522,Z 85,A 146.0247,B 24.8989,C -2.3209,E1 24.8592,E2 298.6216} C_DIS
LIN {X -69.0579,Y 39.205,Z 85,A 144.556,B 24.8989,C -2.3221,E1 24.8612,E2 300.095} C_DIS
LIN {X -68.1184,Y 40.8162,Z 85,A 143.2032,B 24.8985,C -2.3258,E1 24.8631,E2 301.4461} C_DIS
LIN {X -66.8976,Y 42.7854,Z 85,A 141.2925,B 24.8986,C -2.3245,E1 24.866,E2 303.3696} C_DIS
LIN {X -65.3912,Y 45.055,Z 85,A 139.6198,B 24.8975,C -2.3372,E1 24.8686,E2 305.0202} C_DIS
LIN {X -64.0902,Y 46.8861,Z 85,A 137.7963,B 24.8975,C -2.3365,E1 24.8716,E2 306.8543} C_DIS
LIN {X -62.299,Y 49.2411,Z 85,A 135.6367,B 24.8971,C -2.3415,E1 24.8753,E2 309.0123} C_DIS
LIN {X -60.4465,Y 51.4983,Z 85,A 133.5406,B 24.8966,C -2.3472,E1 24.879,E2 311.1044} C_DIS
LIN {X -58.5122,Y 53.686,Z 85,A 131.3067,B 24.8964,C -2.3493,E1 24.8832,E2 313.3433} C_DIS
LIN {X -56.491,Y 55.8088,Z 85,A 129.2717,B 24.8958,C -2.3564,E1 24.8871,E2 315.37} C_DIS
LIN {X -54.3728,Y 57.8745,Z 85,A 127.1407,B 24.8954,C -2.3615,E1 24.8914,E2 317.4977} C_DIS
LIN {X -52.2083,Y 59.8344,Z 85,A 125.0454,B 24.8949,C -2.3666,E1 24.8958,E2 319.5892} C_DIS
LIN {X -49.9732,Y 61.7133,Z 85,A 122.8405,B 24.8947,C -2.3687,E1 24.9005,E2 321.7976} C_DIS
LIN {X -47.5045,Y 63.6336,Z 85,A 120.6488,B 24.8942,C -2.375,E1 24.9054,E2 323.9821} C_DIS
LIN {X -45.6931,Y 64.9476,Z 85,A 119.1401,B 24.8936,C -2.381,E1 24.9088,E2 325.4818} C_DIS
LIN {X -44.0324,Y 66.0844,Z 85,A 117.6801,B 24.8934,C -2.3836,E1 24.9122,E2 326.9403} C_DIS
LIN {X -42.4722,Y 67.0984,Z 85,A 116.1707,B 24.8935,C -2.3818,E1 24.9157,E2 328.459} C_DIS
LIN {X -39.9866,Y 68.6088,Z 85,A 114.1758,B 24.893,C -2.3883,E1 24.9205,E2 330.4444} C_DIS
LIN {X -38.2994,Y 69.5647,Z 85,A 112.7773,B 24.8927,C -2.3907,E1 24.9239,E2 331.8413} C_DIS
LIN {X -35.9409,Y 70.8107,Z 85,A 110.63,B 24.893,C -2.388,E1 24.9293,E2 334.0008} C_DIS
LIN {X -33.0655,Y 72.1995,Z 85,A 108.5258,B 24.8922,C -2.3968,E1 24.9345,E2 336.0894} C_DIS
LIN {X -31.2156,Y 73.0179,Z 85,A 107.1098,B 24.8919,C -2.4001,E1 24.9381,E2 337.501} C_DIS
LIN {X -29.4769,Y 73.7373,Z 85,A 105.7485,B 24.8917,C -2.4019,E1 24.9417,E2 338.8611} C_DIS
LIN {X -27.5645,Y 74.4728,Z 85,A 104.3183,B 24.8914,C -2.4051,E1 24.9454,E2 340.2866} C_DIS
LIN {X -25.8109,Y 75.0991,Z 85,A 102.6979,B 24.892,C -2.3993,E1 24.9497,E2 341.9238} C_DIS
LIN {X -23.0406,Y 75.9948,Z 85,A 100.7648,B 24.8913,C -2.4062,E1 24.9548,E2 343.8439} C_DIS
LIN {X -21.1754,Y 76.5356,Z 85,A 99.244,B 24.8915,C -2.4045,E1 24.9589,E2 345.3713} C_DIS
LIN {X -18.3539,Y 77.2607,Z 85,A 97.2997,B 24.8909,C -2.4107,E1 24.9642,E2 347.3035} C_DIS
LIN {X -16.4592,Y 77.6864,Z 85,A 95.8572,B 24.8909,C -2.4108,E1 24.9681,E2 348.7476} C_DIS
LIN {X -14.48,Y 78.0793,Z 85,A 94.4753,B 24.8906,C -2.414,E1 24.9719,E2 350.1234} C_DIS
LIN {X -12.2806,Y 78.4542,Z 85,A 92.6413,B 24.8911,C -2.4091,E1 24.977,E2 351.9709} C_DIS
LIN {X -9.6333,Y 78.824,Z 85,A 90.9465,B 24.8904,C -2.4166,E1 24.9816,E2 353.649} C_DIS
LIN {X -7.6991,Y 79.0363,Z 85,A 89.5412,B 24.8904,C -2.4173,E1 24.9855,E2 355.0535} C_DIS
LIN {X -5.76,Y 79.2013,Z 85,A 87.9096,B 24.8909,C -2.4117,E1 24.9901,E2 356.6991} C_DIS
LIN {X -2.6563,Y 79.3653,Z 85,A 85.6153,B 24.8909,C -2.411,E1 24.9965,E2 358.9955} C_DIS
LIN {X 0.0599,Y 79.4106,Z 85,A 83.6848,B 24.8909,C -2.4122,E1 25.0019,E2 360.9231} C_DIS
LIN {X 2.882,Y 79.3584,Z 85,A 81.8389,B 24.8903,C -2.4178,E1 25.007,E2 362.7556} C_DIS
LIN {X 5.6909,Y 79.2059,Z 85,A 79.567,B 24.8909,C -2.411,E1 25.0134,E2 365.0426} C_DIS
LIN {X 9.183,Y 78.8767,Z 85,A 77.0979,B 24.8908,C -2.4124,E1 25.0202,E2 367.5067} C_DIS
LIN {X 11.7241,Y 78.5403,Z 85,A 75.3734,B 24.8905,C -2.4154,E1 25.025,E2 369.2225} C_DIS
LIN {X 14.5276,Y 78.0707,Z 85,A 73.3055,B 24.8906,C -2.4142,E1 25.0306,E2 371.2911} C_DIS
LIN {X 16.561,Y 77.6642,Z 85,A 71.9432,B 24.8903,C -2.4174,E1 25.0343,E2 372.6443} C_DIS
LIN {X 18.3707,Y 77.2566,Z 85,A 70.5073,B 24.8907,C -2.4139,E1 25.0383,E2 374.0864} C_DIS
LIN {X 20.703,Y 76.6632,Z 85,A 68.6628,B 24.891,C -2.4097,E1 25.0433,E2 375.9379} C_DIS
LIN {X 23.1347,Y 75.9658,Z 85,A 67.0473,B 24.8906,C -2.4144,E1 25.0476,E2 377.5394} C_DIS
LIN {X 24.9873,Y 75.3768,Z 85,A 65.5952,B 24.8908,C -2.4119,E1 25.0514,E2 378.9949} C_DIS
LIN {X 27.062,Y 74.6561,Z 85,A 63.8357,B 24.8914,C -2.4054,E1 25.0561,E2 380.7661} C_DIS
LIN {X 29.4894,Y 73.7324,Z 85,A 62.1427,B 24.8911,C -2.4088,E1 25.0605,E2 382.4472} C_DIS
LIN {X 31.2875,Y 72.9876,Z 85,A 60.6933,B 24.8914,C -2.406,E1 25.0642,E2 383.8999} C_DIS
LIN {X 33.1369,Y 72.1663,Z 85,A 59.335,B 24.8912,C -2.4074,E1 25.0676,E2 385.2517} C_DIS
LIN {X 34.826,Y 71.3669,Z 85,A 57.6721,B 24.8922,C -2.3965,E1 25.0719,E2 386.9359} C_DIS
LIN {X 37.5114,Y 69.9922,Z 85,A 55.8228,B 24.8916,C -2.4033,E1 25.0764,E2 388.7639} C_DIS
LIN {X 39.213,Y 69.0533,Z 85,A 54.4251,B 24.8918,C -2.4015,E1 25.0798,E2 390.1618} C_DIS
LIN {X 40.8252,Y 68.1131,Z 85,A 52.9781,B 24.8922,C -2.3966,E1 25.0833,E2 391.616} C_DIS
LIN {X 42.4875,Y 67.0888,Z 85,A 51.5574,B 24.8924,C -2.3941,E1 25.0867,E2 393.0381} C_DIS
LIN {X 44.2189,Y 65.9597,Z 85,A 50.1434,B 24.8924,C -2.3941,E1 25.09,E2 394.4476} C_DIS
LIN {X 45.7494,Y 64.9081,Z 85,A 48.8082,B 24.8926,C -2.3919,E1 25.093,E2 395.7831} C_DIS
LIN {X 47.7705,Y 63.4338,Z 85,A 46.9027,B 24.8932,C -2.3858,E1 25.0973,E2 397.6963} C_DIS
LIN {X 49.9987,Y 61.6926,Z 85,A 44.8652,B 24.8935,C -2.3822,E1 25.1018,E2 399.7348} C_DIS
LIN {X 52.2689,Y 59.7814,Z 85,A 42.7229,B 24.8939,C -2.378,E1 25.1063,E2 401.8786} C_DIS
LIN {X 54.4315,Y 57.8193,Z 85,A 40.5426,B 24.8945,C -2.3716,E1 25.1108,E2 404.0653} C_DIS
LIN {X 56.5173,Y 55.7822,Z 85,A 38.536,B 24.8945,C -2.3701,E1 25.1148,E2 406.0669} C_DIS
LIN {X 58.5206,Y 53.6768,Z 85,A 36.4533,B 24.895,C -2.3659,E1 25.1188,E2 408.1504} C_DIS
LIN {X 60.4728,Y 51.4674,Z 85,A 34.3322,B 24.8954,C -2.3613,E1 25.1226,E2 410.2729} C_DIS
LIN {X 62.3042,Y 49.2346,Z 85,A 32.2637,B 24.8958,C -2.3568,E1 25.1263,E2 412.3423} C_DIS
LIN {X 63.8306,Y 47.2406,Z 85,A 30.5719,B 24.8958,C -2.3561,E1 25.1291,E2 414.0277} C_DIS
LIN {X 64.925,Y 45.7256,Z 85,A 29.2068,B 24.8962,C -2.3523,E1 25.1313,E2 415.3953} C_DIS
LIN {X 66.0739,Y 44.0483,Z 85,A 27.7345,B 24.8965,C -2.3484,E1 25.1336,E2 416.8695} C_DIS
LIN {X 67.6461,Y 41.5936,Z 85,A 25.6818,B 24.8969,C -2.3445,E1 25.1367,E2 418.921} C_DIS
LIN {X 68.6051,Y 39.9928,Z 85,A 24.0712,B 24.8979,C -2.3328,E1 25.139,E2 420.551} C_DIS
LIN {X 70.0738,Y 37.3587,Z 85,A 22.1792,B 24.8976,C -2.3357,E1 25.1415,E2 422.4262} C_DIS
LIN {X 70.9682,Y 35.6305,Z 85,A 20.7837,B 24.898,C -2.3321,E1 25.1433,E2 423.8227} C_DIS
LIN {X 71.7873,Y 33.951,Z 85,A 19.4438,B 24.8983,C -2.3286,E1 25.1449,E2 425.1638} C_DIS
LIN {X 72.6287,Y 32.1107,Z 85,A 17.7961,B 24.8991,C -2.3187,E1 25.1468,E2 426.826} C_DIS
LIN {X 73.7348,Y 29.4834,Z 85,A 15.903,B 24.8992,C -2.3178,E1 25.1488,E2 428.7106} C_DIS
LIN {X 74.481,Y 27.542,Z 85,A 14.5154,B 24.8992,C -2.317,E1 25.1502,E2 430.0924} C_DIS
LIN {X 75.1013,Y 25.8042,Z 85,A 12.8698,B 24.9005,C -2.3033,E1 25.1517,E2 431.7612} C_DIS
LIN {X 76.0749,Y 22.7708,Z 85,A 10.6661,B 24.9008,C -2.2994,E1 25.1535,E2 433.9616} C_DIS
LIN {X 76.7796,Y 20.272,Z 85,A 8.972,B 24.9008,C -2.2994,E1 25.1548,E2 435.6461} C_DIS
LIN {X 77.2793,Y 18.2737,Z 85,A 7.5652,B 24.901,C -2.2973,E1 25.1557,E2 437.0496} C_DIS
LIN {X 77.6884,Y 16.45,Z 85,A 6.1288,B 24.9016,C -2.2904,E1 25.1565,E2 438.4939} C_DIS
LIN {X 78.1964,Y 13.8285,Z 85,A 4.1763,B 24.9022,C -2.2836,E1 25.1576,E2 440.4509} C_DIS
LIN {X 78.5517,Y 11.6502,Z 85,A 2.6319,B 24.9025,C -2.2801,E1 25.1582,E2 441.9944} C_DIS
LIN {X 78.8226,Y 9.6445,Z 85,A 1.2805,B 24.9025,C -2.279,E1 25.1587,E2 443.3406} C_DIS
LIN {X 79.0354,Y 7.7097,Z 85,A -0.1157,B 24.9029,C -2.2748,E1 25.1591,E2 444.7383} C_DIS
LIN {X 79.2006,Y 5.7704,Z 85,A -1.7972,B 24.904,C -2.2617,E1 25.1595,E2 446.441} C_DIS
LIN {X 79.3573,Y 2.9166,Z 85,A -3.6067,B 24.904,C -2.2631,E1 25.1597,E2 448.2365} C_DIS
LIN {X 79.4059,Y 0.8414,Z 85,A -4.9874,B 24.904,C -2.262,E1 25.1597,E2 449.6114} C_DIS
LIN {X 79.4035,Y -1.0517,Z 85,A -6.5138,B 24.9048,C -2.2526,E1 25.1597,E2 451.151} C_DIS
LIN {X 79.3113,Y -3.9687,Z 85,A -8.4936,B 24.905,C -2.2498,E1 25.1595,E2 453.1255} C_DIS
LIN {X 79.1903,Y -5.9104,Z 85,A -9.8927,B 24.9054,C -2.2455,E1 25.1593,E2 454.5266} C_DIS
LIN {X 79.0202,Y -7.8633,Z 85,A -11.4023,B 24.906,C -2.2379,E1 25.1589,E2 456.045} C_DIS
LIN {X 78.8011,Y -9.8183,Z 85,A -12.782,B 24.9063,C -2.2347,E1 25.1584,E2 457.4243} C_DIS
LIN {X 78.542,Y -11.7129,Z 85,A -14.1577,B 24.9067,C -2.2304,E1 25.1579,E2 458.802} C_DIS
LIN {X 78.2351,Y -13.6137,Z 85,A -15.5578,B 24.9071,C -2.2256,E1 25.1572,E2 460.2052} C_DIS
LIN {X 77.8655,Y -15.5875,Z 85,A -16.9335,B 24.9073,C -2.2233,E1 25.1565,E2 461.5782} C_DIS
LIN {X 77.3389,Y -18.0159,Z 85,A -18.8181,B 24.908,C -2.2148,E1 25.1554,E2 463.472} C_DIS
LIN {X 76.7639,Y -20.3303,Z 85,A -20.3732,B 24.908,C -2.2146,E1 25.1543,E2 465.0186} C_DIS
LIN {X 76.2444,Y -22.1993,Z 85,A -21.8148,B 24.9085,C -2.2089,E1 25.1532,E2 466.4654} C_DIS
LIN {X 75.703,Y -23.9821,Z 85,A -23.2083,B 24.909,C -2.2031,E1 25.152,E2 467.8646} C_DIS
LIN {X 75.0624,Y -25.9162,Z 85,A -24.5592,B 24.909,C -2.2023,E1 25.1508,E2 469.2098} C_DIS
LIN {X 74.4057,Y -27.7454,Z 85,A -26.0037,B 24.9095,C -2.1967,E1 25.1494,E2 470.6595} C_DIS
LIN {X 73.7336,Y -29.4865,Z 85,A -27.343,B 24.9098,C -2.1928,E1 25.1481,E2 472.0005} C_DIS
LIN {X 72.8947,Y -31.5004,Z 85,A -28.8062,B 24.9099,C -2.1916,E1 25.1465,E2 473.4586} C_DIS
LIN {X 72.1699,Y -33.1291,Z 85,A -30.1397,B 24.9104,C -2.1862,E1 25.1449,E2 474.7975} C_DIS
LIN {X 71.3719,Y -34.8157,Z 85,A -31.5215,B 24.9108,C -2.1811,E1 25.1433,E2 476.1841} C_DIS
LIN {X 70.4979,Y -36.553,Z 85,A -32.9634,B 24.9112,C -2.1757,E1 25.1414,E2 477.6309} C_DIS
LIN {X 69.3913,Y -38.6098,Z 85,A -34.7526,B 24.9119,C -2.1676,E1 25.139,E2 479.43} C_DIS
LIN {X 68.1092,Y -40.8317,Z 85,A -36.4762,B 24.9119,C -2.1662,E1 25.1366,E2 481.1478} C_DIS
LIN {X 67.0884,Y -42.4881,Z 85,A -37.8233,B 24.9122,C -2.1641,E1 25.1346,E2 482.4933} C_DIS
LIN {X 65.9838,Y -44.1832,Z 85,A -39.2743,B 24.9125,C -2.1603,E1 25.1324,E2 483.946} C_DIS
LIN {X 64.9264,Y -45.7237,Z 85,A -40.7093,B 24.913,C -2.1538,E1 25.1301,E2 485.3892} C_DIS
LIN {X 63.7279,Y -47.3789,Z 85,A -42.2547,B 24.9135,C -2.1477,E1 25.1275,E2 486.9418} C_DIS
LIN {X 61.8957,Y -49.7482,Z 85,A -44.3779,B 24.9139,C -2.1431,E1 25.1238,E2 489.0657} C_DIS
LIN {X 60.1294,Y -51.8704,Z 85,A -46.4273,B 24.9144,C -2.1362,E1 25.1201,E2 491.1221} C_DIS
LIN {X 58.1837,Y -54.0439,Z 85,A -48.5258,B 24.9148,C -2.1311,E1 25.1161,E2 493.2234} C_DIS
LIN {X 56.1164,Y -56.1872,Z 85,A -50.635,B 24.9151,C -2.1271,E1 25.112,E2 495.333} C_DIS
LIN {X 54.015,Y -58.2102,Z 85,A -52.7418,B 24.9155,C -2.1221,E1 25.1077,E2 497.4431} C_DIS
LIN {X 51.8406,Y -60.1549,Z 85,A -54.8263,B 24.9159,C -2.1179,E1 25.1034,E2 499.5292} C_DIS
LIN {X 49.5443,Y -62.0594,Z 85,A -56.9413,B 24.9162,C -2.1143,E1 25.0988,E2 501.6446} C_DIS
LIN {X 47.2377,Y -63.8327,Z 85,A -58.9451,B 24.9162,C -2.1128,E1 25.0943,E2 503.6447} C_DIS
LIN {X 44.9879,Y -65.4378,Z 85,A -60.8969,B 24.9165,C -2.1101,E1 25.0899,E2 505.5963} C_DIS
LIN {X 43.2414,Y -66.6048,Z 85,A -62.3037,B 24.9165,C -2.1104,E1 25.0866,E2 506.9976} C_DIS
LIN {X 41.5967,Y -67.6442,Z 85,A -63.7512,B 24.9168,C -2.1065,E1 25.0832,E2 508.4498} C_DIS
LIN {X 39.9941,Y -68.6044,Z 85,A -65.2682,B 24.9174,C -2.0989,E1 25.0795,E2 509.9801} C_DIS
LIN {X 37.4054,Y -70.0493,Z 85,A -67.2698,B 24.9174,C -2.0993,E1 25.0746,E2 511.9748} C_DIS
LIN {X 35.6135,Y -70.9766,Z 85,A -68.6739,B 24.9174,C -2.0985,E1 25.0711,E2 513.3772} C_DIS
LIN {X 33.9375,Y -71.7936,Z 85,A -70.0146,B 24.9176,C -2.0965,E1 25.0677,E2 514.719} C_DIS
LIN {X 32.1003,Y -72.6332,Z 85,A -71.6277,B 24.9181,C -2.0896,E1 25.0636,E2 516.3445} C_DIS
LIN {X 29.4852,Y -73.7341,Z 85,A -73.759,B 24.9185,C -2.0842,E1 25.0581,E2 518.4837} C_DIS
LIN {X 26.7349,Y -74.7751,Z 85,A -75.6221,B 24.9182,C -2.0891,E1 25.0532,E2 520.3313} C_DIS
LIN {X 24.8283,Y -75.4293,Z 85,A -77.0799,B 24.9183,C -2.0872,E1 25.0493,E2 521.7908} C_DIS
LIN {X 22.9836,Y -76.0117,Z 85,A -78.5038,B 24.9185,C -2.0847,E1 25.0455,E2 523.2179} C_DIS
LIN {X 21.1399,Y -76.5451,Z 85,A -79.8423,B 24.9185,C -2.0846,E1 25.0419,E2 524.5545} C_DIS
LIN {X 18.7841,Y -77.1558,Z 85,A -81.7422,B 24.919,C -2.0786,E1 25.0368,E2 526.4658} C_DIS
LIN {X 16.4555,Y -77.6872,Z 85,A -83.3586,B 24.9189,C -2.0801,E1 25.0324,E2 528.0763} C_DIS
LIN {X 14.4517,Y -78.0844,Z 85,A -84.7403,B 24.9187,C -2.0816,E1 25.0286,E2 529.4529} C_DIS
LIN {X 12.5338,Y -78.4151,Z 85,A -86.142,B 24.9188,C -2.0806,E1 25.0247,E2 530.8555} C_DIS
LIN {X 10.6083,Y -78.6987,Z 85,A -87.5961,B 24.919,C -2.0782,E1 25.0207,E2 532.3141} C_DIS
LIN {X 8.1171,Y -78.9936,Z 85,A -89.4703,B 24.9192,C -2.0753,E1 25.0155,E2 534.1938} C_DIS
LIN {X 5.707,Y -79.2049,Z 85,A -91.0637,B 24.919,C -2.0789,E1 25.0111,E2 535.778} C_DIS
LIN {X 3.8124,Y -79.3189,Z 85,A -92.4635,B 24.919,C -2.0774,E1 25.0072,E2 537.1807} C_DIS
LIN {X 1.9454,Y -79.3871,Z 85,A -93.9111,B 24.9193,C -2.0741,E1 25.0031,E2 538.6358} C_DIS
LIN {X 1.9454,Y -79.3871,Z 85,A -93.9111,B 24.9193,C -2.0741,E1 25.0031,E2 538.6358} C_DIS
Enddeposition()
LIN {X 0.5928,Y -88.0077,Z 86,A -94.2661,B 24.9287,C -1.9499,E1 25.0013,E2 539.2854} C_DIS
Startdeposition()
$VEL.CP = VEL_PRINT
LIN {X 3.2395,Y -87.9517,Z 86,A -92.1652,B 24.9278,C -1.9627,E1 25.0072,E2 537.1545} C_DIS
LIN {X 5.3969,Y -87.8457,Z 86,A -90.7603,B 24.9278,C -1.9633,E1 25.0112,E2 535.7489} C_DIS
LIN {X 8.1669,Y -87.6299,Z 86,A -88.8907,B 24.9275,C -1.9662,E1 25.0164,E2 533.8734} C_DIS
LIN {X 10.9697,Y -87.324,Z 86,A -87.2352,B 24.9279,C -1.9614,E1 25.0209,E2 532.2305} C_DIS
LIN {X 12.9486,Y -87.0534,Z 86,A -85.8636,B 24.9276,C -1.9646,E1 25.0248,E2 530.8525} C_DIS
LIN {X 15.0466,Y -86.7156,Z 86,A -84.4613,B 24.9276,C -1.9663,E1 25.0286,E2 529.4477} C_DIS
LIN {X 17.2045,Y -86.3131,Z 86,A -83.0562,B 24.9275,C -1.9667,E1 25.0325,E2 528.0433} C_DIS
LIN {X 19.3175,Y -85.8649,Z 86,A -81.6315,B 24.9273,C -1.9686,E1 25.0364,E2 526.616} C_DIS
LIN {X 21.4783,Y -85.3497,Z 86,A -80.212,B 24.9273,C -1.9691,E1 25.0402,E2 525.1973} C_DIS
LIN {X 23.955,Y -84.6868,Z 86,A -78.3831,B 24.9268,C -1.9763,E1 25.0452,E2 523.3543} C_DIS
LIN {X 26.5799,Y -83.9017,Z 86,A -76.7235,B 24.9269,C -1.9741,E1 25.0496,E2 521.7028} C_DIS
LIN {X 28.664,Y -83.2125,Z 86,A -75.3193,B 24.9269,C -1.9751,E1 25.0533,E2 520.2991} C_DIS
LIN {X 30.6648,Y -82.4964,Z 86,A -73.9395,B 24.9267,C -1.9768,E1 25.0569,E2 518.9182} C_DIS
LIN {X 32.7126,Y -81.7058,Z 86,A -72.5147,B 24.9266,C -1.9786,E1 25.0606,E2 517.4921} C_DIS
LIN {X 34.6757,Y -80.8924,Z 86,A -71.1357,B 24.9265,C -1.9805,E1 25.0642,E2 516.112} C_DIS
LIN {X 36.6505,Y -80.0171,Z 86,A -69.7344,B 24.9263,C -1.9825,E1 25.0677,E2 514.7095} C_DIS
LIN {X 39.0388,Y -78.8776,Z 86,A -67.8727,B 24.9257,C -1.99,E1 25.0725,E2 512.8349} C_DIS
LIN {X 41.519,Y -77.6023,Z 86,A -66.2299,B 24.926,C -1.9871,E1 25.0765,E2 511.2035} C_DIS
LIN {X 43.411,Y -76.56,Z 86,A -64.8289,B 24.9258,C -1.9894,E1 25.0799,E2 509.8011} C_DIS
LIN {X 45.2768,Y -75.4716,Z 86,A -63.4071,B 24.9256,C -1.9925,E1 25.0833,E2 508.3764} C_DIS
LIN {X 47.0858,Y -74.3567,Z 86,A -62.0089,B 24.9253,C -1.9957,E1 25.0866,E2 506.9753} C_DIS
LIN {X 48.9255,Y -73.1591,Z 86,A -60.6278,B 24.9253,C -1.9968,E1 25.0899,E2 505.596} C_DIS
LIN {X 50.6776,Y -71.9567,Z 86,A -59.2049,B 24.9249,C -2.0009,E1 25.0931,E2 504.1682} C_DIS
LIN {X 53.2918,Y -70.0426,Z 86,A -57.1296,B 24.9247,C -2.0042,E1 25.0978,E2 502.0927} C_DIS
LIN {X 55.0219,Y -68.6916,Z 86,A -55.7075,B 24.9245,C -2.007,E1 25.1009,E2 500.6691} C_DIS
LIN {X 56.6911,Y -67.3206,Z 86,A -54.3079,B 24.9243,C -2.0099,E1 25.1039,E2 499.268} C_DIS
LIN {X 58.3001,Y -65.9325,Z 86,A -52.9313,B 24.924,C -2.0129,E1 25.1068,E2 497.89} C_DIS
LIN {X 59.9261,Y -64.4578,Z 86,A -51.5308,B 24.9239,C -2.0152,E1 25.1097,E2 496.4896} C_DIS
LIN {X 61.5298,Y -62.9283,Z 86,A -49.8713,B 24.923,C -2.0262,E1 25.1131,E2 494.8111} C_DIS
LIN {X 63.7419,Y -60.6874,Z 86,A -48.0149,B 24.9231,C -2.0245,E1 25.1166,E2 492.9667} C_DIS
LIN {X 65.2354,Y -59.0787,Z 86,A -46.6355,B 24.9231,C -2.0263,E1 25.1192,E2 491.589} C_DIS
LIN {X 66.6429,Y -57.4866,Z 86,A -45.2386,B 24.9227,C -2.0303,E1 25.1218,E2 490.1889} C_DIS
LIN {X 68.0337,Y -55.8338,Z 86,A -43.8197,B 24.9224,C -2.0345,E1 25.1243,E2 488.7668} C_DIS
LIN {X 69.502,Y -53.9934,Z 86,A -42.4086,B 24.9224,C -2.0343,E1 25.1268,E2 487.3628} C_DIS
LIN {X 70.6913,Y -52.4283,Z 86,A -41.0238,B 24.9219,C -2.0414,E1 25.1291,E2 485.9678} C_DIS
LIN {X 71.9767,Y -50.6489,Z 86,A -39.6087,B 24.9216,C -2.0448,E1 25.1314,E2 484.5515} C_DIS
LIN {X 73.1787,Y -48.8965,Z 86,A -38.2284,B 24.9213,C -2.0485,E1 25.1336,E2 483.1692} C_DIS
LIN {X 74.3567,Y -47.0858,Z 86,A -36.8511,B 24.9211,C -2.0515,E1 25.1356,E2 481.7919} C_DIS
LIN {X 75.5076,Y -45.2167,Z 86,A -35.452,B 24.9208,C -2.0545,E1 25.1377,E2 480.3928} C_DIS
LIN {X 76.5946,Y -43.35,Z 86,A -34.0548,B 24.9206,C -2.0583,E1 25.1396,E2 478.9939} C_DIS
LIN {X 77.619,Y -41.4882,Z 86,A -32.4594,B 24.9197,C -2.0698,E1 25.1418,E2 477.3797} C_DIS
LIN {X 79.1087,Y -38.5716,Z 86,A -30.5411,B 24.9197,C -2.0685,E1 25.1441,E2 475.4746} C_DIS
LIN {X 80.0314,Y -36.6186,Z 86,A -29.1436,B 24.9195,C -2.0724,E1 25.1458,E2 474.0754} C_DIS
LIN {X 80.8924,Y -34.6757,Z 86,A -27.7695,B 24.9192,C -2.0763,E1 25.1473,E2 472.6998} C_DIS
LIN {X 81.7318,Y -32.6475,Z 86,A -26.3501,B 24.9188,C -2.0803,E1 25.1488,E2 471.2787} C_DIS
LIN {X 82.4964,Y -30.6648,Z 86,A -24.9758,B 24.9185,C -2.0842,E1 25.1502,E2 469.9028} C_DIS
LIN {X 83.2241,Y -28.631,Z 86,A -23.5587,B 24.9182,C -2.089,E1 25.1515,E2 468.4825} C_DIS
LIN {X 83.9017,Y -26.5799,Z 86,A -22.1617,B 24.9178,C -2.093,E1 25.1527,E2 467.0839} C_DIS
LIN {X 84.5383,Y -24.4792,Z 86,A -20.6016,B 24.9171,C -2.1022,E1 25.1539,E2 465.5111} C_DIS
LIN {X 85.3737,Y -21.385,Z 86,A -18.6907,B 24.9171,C -2.1025,E1 25.1553,E2 463.6104} C_DIS
LIN {X 85.8803,Y -19.2491,Z 86,A -17.2929,B 24.9168,C -2.1059,E1 25.1561,E2 462.2127} C_DIS
LIN {X 86.4185,Y -16.6596,Z 86,A -15.429,B 24.916,C -2.1165,E1 25.1572,E2 460.3347} C_DIS
LIN {X 86.8937,Y -13.9813,Z 86,A -13.8035,B 24.916,C -2.1169,E1 25.1579,E2 458.7177} C_DIS
LIN {X 87.2422,Y -11.6012,Z 86,A -12.2322,B 24.9155,C -2.1221,E1 25.1585,E2 457.1433} C_DIS
LIN {X 87.5907,Y -8.5917,Z 86,A -10.3107,B 24.9152,C -2.1266,E1 25.1591,E2 455.2226} C_DIS
LIN {X 87.7752,Y -6.4396,Z 86,A -8.9145,B 24.9148,C -2.1308,E1 25.1594,E2 453.8249} C_DIS
LIN {X 87.9068,Y -4.2835,Z 86,A -7.5182,B 24.9145,C -2.1349,E1 25.1596,E2 452.4271} C_DIS
LIN {X 88.0047,Y -1.08,Z 86,A -5.1108,B 24.9131,C -2.153,E1 25.1598,E2 449.9912} C_DIS
LIN {X 87.9837,Y 2.1949,Z 86,A -3.3293,B 24.9135,C -2.1474,E1 25.1598,E2 448.2337} C_DIS
LIN {X 87.9033,Y 4.3535,Z 86,A -1.9325,B 24.9132,C -2.1515,E1 25.1595,E2 446.8354} C_DIS
LIN {X 87.77,Y 6.5094,Z 86,A -0.3115,B 24.9122,C -2.1636,E1 25.1592,E2 445.1956} C_DIS
LIN {X 87.475,Y 9.7008,Z 86,A 1.5572,B 24.9122,C -2.1625,E1 25.1587,E2 443.3406} C_DIS
LIN {X 87.1847,Y 12.0273,Z 86,A 2.9865,B 24.9122,C -2.1638,E1 25.1582,E2 441.9165} C_DIS
LIN {X 86.8879,Y 14.0159,Z 86,A 4.554,B 24.9111,C -2.1771,E1 25.1575,E2 440.3269} C_DIS
LIN {X 86.3131,Y 17.2045,Z 86,A 6.4681,B 24.9111,C -2.1767,E1 25.1565,E2 438.4248} C_DIS
LIN {X 85.8728,Y 19.2834,Z 86,A 7.863,B 24.9107,C -2.1814,E1 25.1557,E2 437.027} C_DIS
LIN {X 85.3737,Y 21.385,Z 86,A 9.2596,B 24.9104,C -2.1853,E1 25.1547,E2 435.6292} C_DIS
LIN {X 84.8232,Y 23.4737,Z 86,A 10.6564,B 24.9101,C -2.1893,E1 25.1537,E2 434.2312} C_DIS
LIN {X 84.2112,Y 25.5818,Z 86,A 12.0342,B 24.9099,C -2.1918,E1 25.1526,E2 432.8554} C_DIS
LIN {X 83.558,Y 27.6407,Z 86,A 13.4314,B 24.9096,C -2.1956,E1 25.1514,E2 431.4569} C_DIS
LIN {X 82.8545,Y 29.683,Z 86,A 14.8287,B 24.9093,C -2.1995,E1 25.1501,E2 430.0584} C_DIS
LIN {X 82.1139,Y 31.6748,Z 86,A 16.4345,B 24.9083,C -2.2113,E1 25.1485,E2 428.4335} C_DIS
LIN {X 80.8784,Y 34.7079,Z 86,A 18.5031,B 24.9079,C -2.2152,E1 25.1463,E2 426.3672} C_DIS
LIN {X 79.7423,Y 37.2407,Z 86,A 20.2315,B 24.9078,C -2.2176,E1 25.1443,E2 424.6426} C_DIS
LIN {X 78.6138,Y 39.5709,Z 86,A 21.8349,B 24.9076,C -2.2193,E1 25.1423,E2 423.0435} C_DIS
LIN {X 77.1041,Y 42.4376,Z 86,A 23.9318,B 24.9072,C -2.2247,E1 25.1395,E2 420.9451} C_DIS
LIN {X 75.9937,Y 44.3944,Z 86,A 25.3134,B 24.9071,C -2.2257,E1 25.1376,E2 419.5683} C_DIS
LIN {X 74.9103,Y 46.1995,Z 86,A 26.7089,B 24.9067,C -2.2301,E1 25.1356,E2 418.1693} C_DIS
LIN {X 73.7539,Y 48.024,Z 86,A 28.1285,B 24.9064,C -2.2342,E1 25.1334,E2 416.7472} C_DIS
LIN {X 72.5732,Y 49.7908,Z 86,A 29.6869,B 24.9056,C -2.2438,E1 25.131,E2 415.1739} C_DIS
LIN {X 70.6703,Y 52.4563,Z 86,A 31.6036,B 24.9057,C -2.2416,E1 25.1278,E2 413.2716} C_DIS
LIN {X 68.7137,Y 54.9947,Z 86,A 33.7004,B 24.9053,C -2.2469,E1 25.1242,E2 411.172} C_DIS
LIN {X 66.9268,Y 57.1534,Z 86,A 35.5913,B 24.9047,C -2.2535,E1 25.1208,E2 409.2743} C_DIS
LIN {X 65.1884,Y 59.1306,Z 86,A 37.2,B 24.9047,C -2.2537,E1 25.1179,E2 407.6723} C_DIS
LIN {X 63.7419,Y 60.6874,Z 86,A 38.7671,B 24.9039,C -2.263,E1 25.1148,E2 406.09} C_DIS
LIN {X 61.6551,Y 62.8046,Z 86,A 40.6364,B 24.9038,C -2.2649,E1 25.1111,E2 404.2242} C_DIS
LIN {X 59.8748,Y 64.5055,Z 86,A 42.0991,B 24.9038,C -2.2633,E1 25.1082,E2 402.7712} C_DIS
LIN {X 58.3001,Y 65.9325,Z 86,A 43.4974,B 24.9036,C -2.2666,E1 25.1053,E2 401.3708} C_DIS
LIN {X 56.6644,Y 67.3434,Z 86,A 44.8979,B 24.9034,C -2.2691,E1 25.1023,E2 399.9698} C_DIS
LIN {X 54.9947,Y 68.7137,Z 86,A 46.3189,B 24.9031,C -2.2722,E1 25.0992,E2 398.5468} C_DIS
LIN {X 53.1196,Y 70.172,Z 86,A 47.7089,B 24.9034,C -2.2697,E1 25.0961,E2 397.1678} C_DIS
LIN {X 51.5283,Y 71.3497,Z 86,A 49.1227,B 24.9028,C -2.2761,E1 25.0929,E2 395.7439} C_DIS
LIN {X 49.6522,Y 72.667,Z 86,A 50.5089,B 24.9028,C -2.275,E1 25.0898,E2 394.3649} C_DIS
LIN {X 47.9948,Y 73.7732,Z 86,A 51.9227,B 24.9024,C -2.281,E1 25.0864,E2 392.9417} C_DIS
LIN {X 46.1698,Y 74.9289,Z 86,A 53.5374,B 24.9016,C -2.2901,E1 25.0826,E2 391.3105} C_DIS
LIN {X 43.35,Y 76.5946,Z 86,A 55.4081,B 24.9021,C -2.2844,E1 25.0781,E2 389.4589} C_DIS
LIN {X 41.4572,Y 77.6354,Z 86,A 57.0594,B 24.9012,C -2.2945,E1 25.074,E2 387.7886} C_DIS
LIN {X 38.6032,Y 79.0935,Z 86,A 58.9327,B 24.9016,C -2.29,E1 25.0694,E2 385.9309} C_DIS
LIN {X 36.6505,Y 80.0171,Z 86,A 60.363,B 24.9014,C -2.2925,E1 25.0657,E2 384.4985} C_DIS
LIN {X 34.4699,Y 80.9791,Z 86,A 61.7279,B 24.9018,C -2.288,E1 25.0623,E2 383.1475} C_DIS
LIN {X 32.6801,Y 81.719,Z 86,A 63.1209,B 24.9013,C -2.2936,E1 25.0586,E2 381.7443} C_DIS
LIN {X 30.6319,Y 82.5084,Z 86,A 64.5254,B 24.9013,C -2.2942,E1 25.055,E2 380.3415} C_DIS
LIN {X 28.631,Y 83.2241,Z 86,A 65.9277,B 24.9011,C -2.296,E1 25.0513,E2 378.9377} C_DIS
LIN {X 26.5799,Y 83.9017,Z 86,A 67.3528,B 24.9009,C -2.2977,E1 25.0475,E2 377.5112} C_DIS
LIN {X 24.4792,Y 84.5383,Z 86,A 68.7371,B 24.9009,C -2.2973,E1 25.0438,E2 376.1303} C_DIS
LIN {X 22.3971,Y 85.1136,Z 86,A 70.1411,B 24.9009,C -2.2981,E1 25.04,E2 374.7265} C_DIS
LIN {X 20.3357,Y 85.6297,Z 86,A 71.6488,B 24.9005,C -2.303,E1 25.0359,E2 373.2096} C_DIS
LIN {X 18.2018,Y 86.1084,Z 86,A 72.9713,B 24.9007,C -2.3004,E1 25.0323,E2 371.895} C_DIS
LIN {X 16.0751,Y 86.5306,Z 86,A 74.3553,B 24.9007,C -2.3001,E1 25.0285,E2 370.5133} C_DIS
LIN {X 12.9139,Y 87.0587,Z 86,A 76.4826,B 24.9006,C -2.302,E1 25.0226,E2 368.3835} C_DIS
LIN {X 10.7387,Y 87.3535,Z 86,A 77.8901,B 24.9006,C -2.3016,E1 25.0187,E2 366.978} C_DIS
LIN {X 8.5917,Y 87.5907,Z 86,A 79.2749,B 24.9006,C -2.3011,E1 25.0149,E2 365.5953} C_DIS
LIN {X 6.3838,Y 87.779,Z 86,A 80.6833,B 24.9007,C -2.3001,E1 25.011,E2 364.19} C_DIS
LIN {X 4.2835,Y 87.9068,Z 86,A 82.087,B 24.9007,C -2.3012,E1 25.0071,E2 362.7843} C_DIS
LIN {X 2.1249,Y 87.9854,Z 86,A 83.5148,B 24.9006,C -2.3017,E1 25.0031,E2 361.3555} C_DIS
LIN {X 0,Y 88.0113,Z 86,A 84.8991,B 24.9006,C -2.3015,E1 24.9992,E2 359.9719} C_DIS
LIN {X -2.1949,Y 87.9837,Z 86,A 86.436,B 24.9004,C -2.3046,E1 24.9949,E2 358.4276} C_DIS
LIN {X -4.3535,Y 87.9033,Z 86,A 87.7148,B 24.9007,C -2.3001,E1 24.9914,E2 357.1592} C_DIS
LIN {X -6.5094,Y 87.77,Z 86,A 89.1224,B 24.9007,C -2.2995,E1 24.9875,E2 355.7523} C_DIS
LIN {X -8.6615,Y 87.5838,Z 86,A 90.5301,B 24.9008,C -2.2989,E1 24.9835,E2 354.3455} C_DIS
LIN {X -10.7735,Y 87.3494,Z 86,A 91.9574,B 24.9008,C -2.2995,E1 24.9796,E2 352.9158} C_DIS
LIN {X -13.0284,Y 87.041,Z 86,A 93.3732,B 24.9011,C -2.2965,E1 24.9757,E2 351.5059} C_DIS
LIN {X -15.0811,Y 86.7094,Z 86,A 94.7551,B 24.9011,C -2.2964,E1 24.9719,E2 350.123} C_DIS
LIN {X -17.2045,Y 86.3131,Z 86,A 96.1636,B 24.9011,C -2.2953,E1 24.968,E2 348.7154} C_DIS
LIN {X -19.3175,Y 85.8649,Z 86,A 97.5939,B 24.9011,C -2.2949,E1 24.9641,E2 347.2845} C_DIS
LIN {X -21.385,Y 85.3737,Z 86,A 98.9803,B 24.9013,C -2.2936,E1 24.9603,E2 345.8991} C_DIS
LIN {X -23.4737,Y 84.8232,Z 86,A 100.4165,B 24.9013,C -2.2931,E1 24.9565,E2 344.4619} C_DIS
LIN {X -25.6167,Y 84.2003,Z 86,A 102.0452,B 24.901,C -2.2969,E1 24.9521,E2 342.8213} C_DIS
LIN {X -28.664,Y 83.2125,Z 86,A 103.9367,B 24.9017,C -2.2885,E1 24.9471,E2 340.9464} C_DIS
LIN {X -30.6648,Y 82.4964,Z 86,A 105.3244,B 24.9019,C -2.2869,E1 24.9435,E2 339.5599} C_DIS
LIN {X -32.7126,Y 81.7058,Z 86,A 106.8721,B 24.9017,C -2.2885,E1 24.9394,E2 338.0048} C_DIS
LIN {X -34.7079,Y 80.8784,Z 86,A 108.1473,B 24.9023,C -2.2826,E1 24.9362,E2 336.7409} C_DIS
LIN {X -36.6505,Y 80.0171,Z 86,A 109.5562,B 24.9023,C -2.2813,E1 24.9326,E2 335.3316} C_DIS
LIN {X -38.6032,Y 79.0935,Z 86,A 110.988,B 24.9025,C -2.2799,E1 24.929,E2 333.8995} C_DIS
LIN {X -40.5636,Y 78.106,Z 86,A 112.4018,B 24.9027,C -2.2771,E1 24.9255,E2 332.4885} C_DIS
LIN {X -42.4416,Y 77.1019,Z 86,A 113.8112,B 24.9029,C -2.2754,E1 24.922,E2 331.0791} C_DIS
LIN {X -44.3171,Y 76.0394,Z 86,A 115.2227,B 24.9031,C -2.2732,E1 24.9186,E2 329.6687} C_DIS
LIN {X -46.1698,Y 74.9289,Z 86,A 116.6139,B 24.9033,C -2.2702,E1 24.9153,E2 328.2803} C_DIS
LIN {X -48.024,Y 73.7539,Z 86,A 118.049,B 24.9035,C -2.2677,E1 24.9119,E2 326.8466} C_DIS
LIN {X -49.7908,Y 72.5732,Z 86,A 119.5353,B 24.9035,C -2.268,E1 24.9085,E2 325.3545} C_DIS
LIN {X -51.5851,Y 71.3087,Z 86,A 120.8525,B 24.904,C -2.2618,E1 24.9055,E2 324.0475} C_DIS
LIN {X -53.2918,Y 70.0426,Z 86,A 122.2846,B 24.9041,C -2.2604,E1 24.9023,E2 322.6137} C_DIS
LIN {X -55.0219,Y 68.6916,Z 86,A 123.6997,B 24.9044,C -2.2569,E1 24.8992,E2 321.2016} C_DIS
LIN {X -56.6911,Y 67.3206,Z 86,A 125.2567,B 24.9044,C -2.2583,E1 24.8959,E2 319.6353} C_DIS
LIN {X -59.2588,Y 65.0707,Z 86,A 127.2193,B 24.9054,C -2.2456,E1 24.8918,E2 317.6952} C_DIS
LIN {X -60.8996,Y 63.5374,Z 86,A 128.6649,B 24.9057,C -2.2417,E1 24.8889,E2 316.253} C_DIS
LIN {X -62.258,Y 62.2085,Z 86,A 130.0597,B 24.9056,C -2.2434,E1 24.8861,E2 314.8483} C_DIS
LIN {X -63.7659,Y 60.6618,Z 86,A 131.4736,B 24.9059,C -2.2402,E1 24.8834,E2 313.436} C_DIS
LIN {X -65.3972,Y 58.898,Z 86,A 132.905,B 24.9065,C -2.2324,E1 24.8807,E2 312.0168} C_DIS
LIN {X -66.784,Y 57.321,Z 86,A 134.5987,B 24.906,C -2.2385,E1 24.8776,E2 310.3009} C_DIS
LIN {X -68.7354,Y 54.9672,Z 86,A 136.419,B 24.9069,C -2.2283,E1 24.8744,E2 308.4964} C_DIS
LIN {X -70.6913,Y 52.4283,Z 86,A 138.5431,B 24.9072,C -2.2239,E1 24.8708,E2 306.3728} C_DIS
LIN {X -71.9767,Y 50.6489,Z 86,A 140.0125,B 24.9075,C -2.2212,E1 24.8684,E2 304.9025} C_DIS
LIN {X -73.4278,Y 48.5187,Z 86,A 141.7886,B 24.9076,C -2.2194,E1 24.8656,E2 303.1218} C_DIS
LIN {X -74.9471,Y 46.1399,Z 86,A 143.4758,B 24.9084,C -2.2099,E1 24.8632,E2 301.4488} C_DIS
LIN {X -76.0394,Y 44.3171,Z 86,A 144.9102,B 24.9086,C -2.2074,E1 24.8611,E2 300.0129} C_DIS
LIN {X -77.1041,Y 42.4376,Z 86,A 146.305,B 24.909,C -2.203,E1 24.8592,E2 298.6213} C_DIS
LIN {X -78.1383,Y 40.5014,Z 86,A 147.7218,B 24.9093,C -2.1985,E1 24.8574,E2 297.2077} C_DIS
LIN {X -79.1087,Y 38.5716,Z 86,A 149.1583,B 24.9096,C -2.1952,E1 24.8556,E2 295.7713} C_DIS
LIN {X -80.0314,Y 36.6186,Z 86,A 150.5531,B 24.91,C -2.1907,E1 24.854,E2 294.3797} C_DIS
LIN {X -80.8924,Y 34.6757,Z 86,A 151.9668,B 24.9103,C -2.1874,E1 24.8524,E2 292.966} C_DIS
LIN {X -81.9184,Y 32.1726,Z 86,A 153.8477,B 24.9104,C -2.1855,E1 24.8504,E2 291.0791} C_DIS
LIN {X -82.8781,Y 29.617,Z 86,A 155.6809,B 24.9107,C -2.1817,E1 24.8487,E2 289.2447} C_DIS
LIN {X -83.9017,Y 26.5799,Z 86,A 157.6511,B 24.9115,C -2.1719,E1 24.847,E2 287.2866} C_DIS
LIN {X -84.5383,Y 24.4792,Z 86,A 159.0691,B 24.9119,C -2.1671,E1 24.8458,E2 285.8718} C_DIS
LIN {X -85.3737,Y 21.385,Z 86,A 161.1912,B 24.9124,C -2.1616,E1 24.8443,E2 283.7506} C_DIS
LIN {X -85.8728,Y 19.2834,Z 86,A 162.5866,B 24.9128,C -2.1568,E1 24.8435,E2 282.3583} C_DIS
LIN {X -86.3268,Y 17.1357,Z 86,A 164.0041,B 24.9131,C -2.152,E1 24.8427,E2 280.9441} C_DIS
LIN {X -86.7156,Y 15.0466,Z 86,A 165.4586,B 24.9133,C -2.1496,E1 24.842,E2 279.4866} C_DIS
LIN {X -87.0587,Y 12.9139,Z 86,A 167.0537,B 24.9133,C -2.1505,E1 24.8413,E2 277.8798} C_DIS
LIN {X -87.475,Y 9.7008,Z 86,A 168.98,B 24.9142,C -2.1385,E1 24.8406,E2 275.9706} C_DIS
LIN {X -87.6868,Y 7.5511,Z 86,A 170.399,B 24.9146,C -2.1344,E1 24.8403,E2 274.5529} C_DIS
LIN {X -87.8567,Y 5.1978,Z 86,A 172.0996,B 24.9146,C -2.1342,E1 24.84,E2 272.8425} C_DIS
LIN {X -87.9901,Y 1.8731,Z 86,A 173.9646,B 24.9158,C -2.1187,E1 24.8398,E2 271.0034} C_DIS
LIN {X -88.0047,Y -1.08,Z 86,A 176.0612,B 24.9159,C -2.1175,E1 24.8398,E2 268.8969} C_DIS
LIN {X -87.9517,Y -3.2395,Z 86,A 177.4775,B 24.9162,C -2.1133,E1 24.8399,E2 267.4821} C_DIS
LIN {X -87.8457,Y -5.3969,Z 86,A 178.8936,B 24.9166,C -2.1091,E1 24.8402,E2 266.0675} C_DIS
LIN {X -87.5838,Y -8.6615,Z 86,A -179.0015,B 24.9172,C -2.1016,E1 24.8407,E2 263.9679} C_DIS
LIN {X -87.3494,Y -10.7735,Z 86,A -177.566,B 24.9174,C -2.0988,E1 24.8411,E2 262.5306} C_DIS
LIN {X -87.0534,Y -12.9486,Z 86,A -176.1692,B 24.9178,C -2.0934,E1 24.8417,E2 261.1383} C_DIS
LIN {X -86.7156,Y -15.0466,Z 86,A -174.7548,B 24.9181,C -2.0899,E1 24.8423,E2 259.7237} C_DIS
LIN {X -86.3131,Y -17.2045,Z 86,A -173.3375,B 24.9185,C -2.0852,E1 24.8431,E2 258.3093} C_DIS
LIN {X -85.8649,Y -19.3175,Z 86,A -171.6883,B 24.9182,C -2.0879,E1 24.8441,E2 256.644} C_DIS
LIN {X -85.1049,Y -22.4311,Z 86,A -169.7994,B 24.9192,C -2.0758,E1 24.8454,E2 254.7729} C_DIS
LIN {X -84.5287,Y -24.5129,Z 86,A -168.3632,B 24.9195,C -2.0725,E1 24.8465,E2 253.3364} C_DIS
LIN {X -83.9017,Y -26.5799,Z 86,A -166.9475,B 24.9198,C -2.0685,E1 24.8476,E2 251.9219} C_DIS
LIN {X -83.0611,Y -29.0956,Z 86,A -165.1044,B 24.9198,C -2.0668,E1 24.8493,E2 250.0723} C_DIS
LIN {X -82.0205,Y -31.9126,Z 86,A -163.1399,B 24.9203,C -2.0614,E1 24.8513,E2 248.1097} C_DIS
LIN {X -80.8924,Y -34.6757,Z 86,A -161.307,B 24.921,C -2.0526,E1 24.8532,E2 246.2876} C_DIS
LIN {X -80.0171,Y -36.6505,Z 86,A -159.8922,B 24.9213,C -2.0489,E1 24.8548,E2 244.8739} C_DIS
LIN {X -79.0779,Y -38.6346,Z 86,A -158.4755,B 24.9216,C -2.0446,E1 24.8565,E2 243.4599} C_DIS
LIN {X -78.106,Y -40.5636,Z 86,A -156.8762,B 24.9215,C -2.0464,E1 24.8586,E2 241.8478} C_DIS
LIN {X -76.56,Y -43.411,Z 86,A -154.9386,B 24.9223,C -2.0357,E1 24.8612,E2 239.9255} C_DIS
LIN {X -75.4716,Y -45.2768,Z 86,A -153.5028,B 24.9225,C -2.0328,E1 24.8632,E2 238.489} C_DIS
LIN {X -74.3567,Y -47.0858,Z 86,A -152.0906,B 24.9227,C -2.0301,E1 24.8653,E2 237.0762} C_DIS
LIN {X -73.1591,Y -48.9255,Z 86,A -150.6958,B 24.9231,C -2.0255,E1 24.8675,E2 235.6854} C_DIS
LIN {X -71.8536,Y -50.8221,Z 86,A -149.2506,B 24.9235,C -2.0201,E1 24.8698,E2 234.2458} C_DIS
LIN {X -70.6239,Y -52.5181,Z 86,A -147.8642,B 24.9237,C -2.0175,E1 24.8721,E2 232.8591} C_DIS
LIN {X -69.3834,Y -54.1473,Z 86,A -146.4349,B 24.9237,C -2.0171,E1 24.8745,E2 231.4238} C_DIS
LIN {X -68.0113,Y -55.8607,Z 86,A -145.0191,B 24.924,C -2.0134,E1 24.877,E2 230.0103} C_DIS
LIN {X -66.6199,Y -57.513,Z 86,A -143.6274,B 24.9243,C -2.0098,E1 24.8795,E2 228.6209} C_DIS
LIN {X -65.2121,Y -59.1048,Z 86,A -141.9965,B 24.9239,C -2.0141,E1 24.8826,E2 226.9725} C_DIS
LIN {X -62.9678,Y -61.4899,Z 86,A -140.0948,B 24.9248,C -2.0026,E1 24.8862,E2 225.0899} C_DIS
LIN {X -61.4398,Y -63.0167,Z 86,A -138.682,B 24.925,C -1.9998,E1 24.889,E2 223.6777} C_DIS
LIN {X -59.8748,Y -64.5055,Z 86,A -137.2478,B 24.9252,C -1.9978,E1 24.892,E2 222.2424} C_DIS
LIN {X -57.4866,Y -66.6429,Z 86,A -135.1524,B 24.9254,C -1.994,E1 24.8963,E2 220.1478} C_DIS
LIN {X -55.3995,Y -68.3856,Z 86,A -133.2534,B 24.9254,C -1.9947,E1 24.9005,E2 218.24} C_DIS
LIN {X -53.2638,Y -70.0637,Z 86,A -131.3965,B 24.9254,C -1.9942,E1 24.9046,E2 216.3774} C_DIS
LIN {X -50.6489,Y -71.9767,Z 86,A -129.5037,B 24.9262,C -1.9841,E1 24.9088,E2 214.5023} C_DIS
LIN {X -48.8965,Y -73.1787,Z 86,A -128.0736,B 24.9262,C -1.9833,E1 24.9121,E2 213.0692} C_DIS
LIN {X -47.0858,Y -74.3567,Z 86,A -126.683,B 24.9264,C -1.9807,E1 24.9154,E2 211.6805} C_DIS
LIN {X -45.2167,Y -75.5076,Z 86,A -125.2706,B 24.9266,C -1.9781,E1 24.9188,E2 210.2699} C_DIS
LIN {X -43.35,Y -76.5946,Z 86,A -123.8601,B 24.9268,C -1.9762,E1 24.9222,E2 208.8595} C_DIS
LIN {X -41.4882,Y -77.619,Z 86,A -122.4309,B 24.9268,C -1.9758,E1 24.9257,E2 207.4273} C_DIS
LIN {X -39.5709,Y -78.6138,Z 86,A -120.8932,B 24.9266,C -1.9781,E1 24.9296,E2 205.8799} C_DIS
LIN {X -36.6186,Y -80.0314,Z 86,A -118.6762,B 24.9266,C -1.9783,E1 24.9352,E2 203.6569} C_DIS
LIN {X -33.6805,Y -81.3118,Z 86,A -116.7915,B 24.9272,C -1.9698,E1 24.94,E2 201.788} C_DIS
LIN {X -31.6421,Y -82.1263,Z 86,A -115.3848,B 24.9274,C -1.9678,E1 24.9436,E2 200.3831} C_DIS
LIN {X -29.6501,Y -82.8665,Z 86,A -113.9937,B 24.9274,C -1.9668,E1 24.9473,E2 198.9916} C_DIS
LIN {X -27.5742,Y -83.58,Z 86,A -112.3386,B 24.927,C -1.9728,E1 24.9517,E2 197.3191} C_DIS
LIN {X -24.4792,Y -84.5383,Z 86,A -110.4497,B 24.9277,C -1.9644,E1 24.9567,E2 195.4471} C_DIS
LIN {X -21.385,Y -85.3737,Z 86,A -108.3602,B 24.9277,C -1.9632,E1 24.9624,E2 193.3572} C_DIS
LIN {X -19.2491,Y -85.8803,Z 86,A -106.9512,B 24.9278,C -1.9619,E1 24.9662,E2 191.9495} C_DIS
LIN {X -16.7077,Y -86.4092,Z 86,A -105.0874,B 24.9275,C -1.9668,E1 24.9713,E2 190.072} C_DIS
LIN {X -13.9813,Y -86.8937,Z 86,A -103.4345,B 24.9279,C -1.9614,E1 24.9759,E2 188.4302} C_DIS
LIN {X -11.8099,Y -87.2151,Z 86,A -102.0047,B 24.9279,C -1.9611,E1 24.9798,E2 187} C_DIS
LIN {X -9.1795,Y -87.5296,Z 86,A -100.1652,B 24.9276,C -1.9646,E1 24.9849,E2 185.151} C_DIS
LIN {X -6.4396,Y -87.7752,Z 86,A -98.5096,B 24.928,C -1.9602,E1 24.9895,E2 183.5053} C_DIS
LIN {X -4.2835,Y -87.9068,Z 86,A -97.0583,B 24.9278,C -1.9617,E1 24.9936,E2 182.0499} C_DIS
LIN {X -2.1249,Y -87.9854,Z 86,A -95.6766,B 24.9278,C -1.9611,E1 24.9974,E2 180.6694} C_DIS
LIN {X 0.5928,Y -88.0077,Z 86,A -94.2663,B 24.9287,C -1.9498,E1 25.0013,E2 179.2859} C_DIS
Enddeposition()
LIN {X 0.5928,Y -88.0077,Z 86,A -94.2663,B 24.9287,C -1.9498,E1 25.0013,E2 179.2859} C_DIS
Startdeposition()
$VEL.CP = VEL_PRINT
LIN {X -0.7859,Y -87.0994,Z 86,A -95.6312,B 24.9287,C -1.9508,E1 24.9975,E2 180.6484} C_DIS
LIN {X -3.8929,Y -87.0156,Z 86,A -97.6911,B 24.9287,C -1.9501,E1 24.9917,E2 182.7103} C_DIS
LIN {X -6.3723,Y -86.8706,Z 86,A -99.3038,B 24.9287,C -1.9507,E1 24.9872,E2 184.3222} C_DIS
LIN {X -9.435,Y -86.5908,Z 86,A -101.2093,B 24.9284,C -1.9546,E1 24.982,E2 186.2195} C_DIS
LIN {X -12.3994,Y -86.2156,Z 86,A -103.2209,B 24.9284,C -1.9535,E1 24.9764,E2 188.2351} C_DIS
LIN {X -14.5789,Y -85.8741,Z 86,A -104.8945,B 24.9289,C -1.947,E1 24.9717,E2 189.9258} C_DIS
LIN {X -17.8411,Y -85.2564,Z 86,A -107.0137,B 24.9287,C -1.9499,E1 24.9659,E2 192.0406} C_DIS
LIN {X -21.8423,Y -84.3196,Z 86,A -109.7522,B 24.9287,C -1.9503,E1 24.9585,E2 194.7819} C_DIS
LIN {X -24.5408,Y -83.5743,Z 86,A -111.6499,B 24.9287,C -1.9498,E1 24.9534,E2 196.6839} C_DIS
LIN {X -28.4471,Y -82.3267,Z 86,A -114.2289,B 24.9283,C -1.9555,E1 24.9466,E2 199.2541} C_DIS
LIN {X -31.5218,Y -81.1994,Z 86,A -116.1166,B 24.9276,C -1.9656,E1 24.9417,E2 201.1217} C_DIS
LIN {X -33.9537,Y -80.2123,Z 86,A -118.3159,B 24.9285,C -1.953,E1 24.9359,E2 203.3559} C_DIS
LIN {X -37.6327,Y -78.5535,Z 86,A -120.7841,B 24.9279,C -1.9617,E1 24.9297,E2 205.8098} C_DIS
LIN {X -40.8317,Y -76.9396,Z 86,A -122.8881,B 24.9271,C -1.9722,E1 24.9246,E2 207.8942} C_DIS
LIN {X -44.7543,Y -74.7273,Z 86,A -126.193,B 24.9275,C -1.9661,E1 24.9165,E2 211.2236} C_DIS
LIN {X -47.088,Y -73.2774,Z 86,A -127.8482,B 24.927,C -1.9734,E1 24.9126,E2 212.8668} C_DIS
LIN {X -49.6986,Y -71.5326,Z 86,A -129.9522,B 24.9268,C -1.9755,E1 24.9078,E2 214.9726} C_DIS
LIN {X -52.3086,Y -69.6467,Z 86,A -132.0918,B 24.9266,C -1.9785,E1 24.9029,E2 217.1126} C_DIS
LIN {X -55.1752,Y -67.3998,Z 86,A -134.4862,B 24.9263,C -1.9829,E1 24.8977,E2 219.5056} C_DIS
LIN {X -57.4082,Y -65.5071,Z 86,A -136.3177,B 24.9258,C -1.9894,E1 24.8939,E2 221.3288} C_DIS
LIN {X -59.6341,Y -63.4872,Z 86,A -138.4996,B 24.9259,C -1.9873,E1 24.8893,E2 223.5244} C_DIS
LIN {X -61.9721,Y -61.2072,Z 86,A -140.578,B 24.9255,C -1.9939,E1 24.8852,E2 225.596} C_DIS
LIN {X -63.9434,Y -59.1458,Z 86,A -142.2546,B 24.9247,C -2.0037,E1 24.8821,E2 227.2564} C_DIS
LIN {X -65.7698,Y -57.1074,Z 86,A -144.3683,B 24.9251,C -1.9987,E1 24.8781,E2 229.3916} C_DIS
LIN {X -68.0849,Y -54.3274,Z 86,A -146.4469,B 24.924,C -2.0129,E1 24.8745,E2 231.4459} C_DIS
LIN {X -69.7071,Y -52.2283,Z 86,A -148.2404,B 24.9238,C -2.0157,E1 24.8714,E2 233.2412} C_DIS
LIN {X -71.3764,Y -49.9232,Z 86,A -150.2819,B 24.9238,C -2.0155,E1 24.8681,E2 235.2934} C_DIS
LIN {X -72.9755,Y -47.5568,Z 86,A -152.28,B 24.9238,C -2.0168,E1 24.865,E2 237.2982} C_DIS
LIN {X -74.8615,Y -44.5272,Z 86,A -154.245,B 24.9224,C -2.0339,E1 24.8622,E2 239.2326} C_DIS
LIN {X -76.1303,Y -42.321,Z 86,A -156.2629,B 24.9228,C -2.0285,E1 24.8594,E2 241.2739} C_DIS
LIN {X -77.3684,Y -40.0146,Z 86,A -157.7605,B 24.922,C -2.0396,E1 24.8574,E2 242.753} C_DIS
LIN {X -78.2106,Y -38.3418,Z 86,A -159.3396,B 24.9225,C -2.0331,E1 24.8555,E2 244.356} C_DIS
LIN {X -79.7798,Y -34.9581,Z 86,A -161.6427,B 24.9216,C -2.0443,E1 24.8528,E2 246.6451} C_DIS
LIN {X -81.0092,Y -32.0062,Z 86,A -163.7731,B 24.9212,C -2.0496,E1 24.8506,E2 248.7748} C_DIS
LIN {X -82.1717,Y -28.8906,Z 86,A -166.0588,B 24.9209,C -2.0532,E1 24.8484,E2 251.0647} C_DIS
LIN {X -83.1857,Y -25.8263,Z 86,A -168.1883,B 24.9205,C -2.0594,E1 24.8466,E2 253.1918} C_DIS
LIN {X -83.9402,Y -23.2627,Z 86,A -170.0171,B 24.9202,C -2.0626,E1 24.8452,E2 255.0234} C_DIS
LIN {X -84.8232,Y -19.7967,Z 86,A -172.3044,B 24.9195,C -2.0717,E1 24.8437,E2 257.3024} C_DIS
LIN {X -85.529,Y -16.4816,Z 86,A -174.6058,B 24.9191,C -2.0765,E1 24.8424,E2 259.6058} C_DIS
LIN {X -86.021,Y -13.6888,Z 86,A -176.4801,B 24.9187,C -2.0821,E1 24.8415,E2 261.478} C_DIS
LIN {X -86.4064,Y -10.9926,Z 86,A -178.5485,B 24.9189,C -2.08,E1 24.8408,E2 263.5638} C_DIS
LIN {X -86.8178,Y -7.0382,Z 86,A 178.4921,B 24.9189,C -2.0788,E1 24.8401,E2 266.5439} C_DIS
LIN {X -87.0417,Y -3.2867,Z 86,A 176.8364,B 24.9166,C -2.1092,E1 24.8399,E2 268.1368} C_DIS
LIN {X -87.0866,Y 1.6669,Z 86,A 173.4614,B 24.916,C -2.1164,E1 24.8399,E2 271.5151} C_DIS
LIN {X -87.0103,Y 4.0184,Z 86,A 171.2915,B 24.917,C -2.1041,E1 24.8401,E2 273.7274} C_DIS
LIN {X -86.7965,Y 7.3026,Z 86,A 169.1096,B 24.9165,C -2.1105,E1 24.8406,E2 275.907} C_DIS
LIN {X -86.4545,Y 10.6166,Z 86,A 167.5905,B 24.9144,C -2.1361,E1 24.8411,E2 277.3741} C_DIS
LIN {X -86.105,Y 13.1459,Z 86,A 165.6587,B 24.9146,C -2.1345,E1 24.8419,E2 279.3214} C_DIS
LIN {X -85.6327,Y 15.943,Z 86,A 163.766,B 24.9141,C -2.1396,E1 24.8428,E2 281.213} C_DIS
LIN {X -84.9419,Y 19.2831,Z 86,A 161.8719,B 24.9128,C -2.1565,E1 24.8439,E2 283.0779} C_DIS
LIN {X -84.3385,Y 21.7687,Z 86,A 159.8807,B 24.913,C -2.1532,E1 24.8453,E2 285.0888} C_DIS
LIN {X -83.468,Y 24.8992,Z 86,A 157.8452,B 24.9123,C -2.1627,E1 24.8468,E2 287.1133} C_DIS
LIN {X -82.79,Y 27.0693,Z 86,A 156.0148,B 24.9127,C -2.158,E1 24.8484,E2 288.9654} C_DIS
LIN {X -81.3561,Y 31.1147,Z 86,A 153.5407,B 24.9112,C -2.1764,E1 24.8508,E2 291.4096} C_DIS
LIN {X -80.4438,Y 33.4046,Z 86,A 151.6605,B 24.9113,C -2.1741,E1 24.8528,E2 293.3058} C_DIS
LIN {X -78.7896,Y 37.138,Z 86,A 148.7358,B 24.9113,C -2.1755,E1 24.8562,E2 296.2432} C_DIS
Enddeposition()
END
